	W =  90.000 deg,	P =   0.000 deg,	R =   90.000 deg
};
P[2097]{
   GP1:
	UF : 0, UT : 6,		CONFIG : 'N U T, 0, 0, 0',
	X =  98.445  mm,	Y =   -678.534  mm,	Z =   -242.195  mm,
	W =  90.000 deg,	P =   0.000 deg,	R =   90.000 deg
};
P[2098]{
   GP1:
	UF : 0, UT : 6,		CONFIG : 'N U T, 0, 0, 0',
	X =  104.284  mm,	Y =   -675.249  mm,	Z =   -241.987  mm,
	W =  90.000 deg,	P =   0.000 deg,	R =   90.000 deg
};
P[2099]{
   GP1:
	UF : 0, UT : 6,		CONFIG : 'N U T, 0, 0, 0',
	X =  105.353  mm,	Y =   -674.513  mm,	Z =   -242.274  mm,
	W =  90.000 deg,	P =   0.000 deg,	R =   90.000 deg
};
P[2100]{
   GP1:
	UF : 0, UT : 6,		CONFIG : 'N U T, 0, 0, 0',
	X =  107.366  mm,	Y =   -673.374  mm,	Z =   -242.215  mm,
	W =  90.000 deg,	P =   0.000 deg,	R =   90.000 deg
};
P[2101]{
   GP1:
	UF : 0, UT : 6,		CONFIG : 'N U T, 0, 0, 0',
	X =  110.303  mm,	Y =   -671.720  mm,	Z =   -242.116  mm,
	W =  90.000 deg,	P =   0.000 deg,	R =   90.000 deg
};
P[2102]{
   GP1:
	UF : 0, UT : 6,		CONFIG : 'N U T, 0, 0, 0',
	X =  111.391  mm,	Y =   -671.119  mm,	Z =   -242.049  mm,
	W =  90.000 deg,	P =   0.000 deg,	R =   90.000 deg
};
P[2103]{
   GP1:
	UF : 0, UT : 6,		CONFIG : 'N U T, 0, 0, 0',
	X =  113.149  mm,	Y =   -670.072  mm,	Z =   -242.125  mm,
	W =  90.000 deg,	P =   0.000 deg,	R =   90.000 deg
};
P[2104]{
   GP1:
	UF : 0, UT : 6,		CONFIG : 'N U T, 0, 0, 0',
	X =  114.405  mm,	Y =   -669.261  mm,	Z =   -242.337  mm,
	W =  90.000 deg,	P =   0.000 deg,	R =   90.000 deg
};
P[2105]{
   GP1:
	UF : 0, UT : 6,		CONFIG : 'N U T, 0, 0, 0',
	X =  118.642  mm,	Y =   -666.812  mm,	Z =   -242.340  mm,
	W =  90.000 deg,	P =   0.000 deg,	R =   90.000 deg
};
P[2106]{
   GP1:
	UF : 0, UT : 6,		CONFIG : 'N U T, 0, 0, 0',
	X =  119.817  mm,	Y =   -666.137  mm,	Z =   -242.334  mm,
	W =  90.000 deg,	P =   0.000 deg,	R =   90.000 deg
};
P[2107]{
   GP1:
	UF : 0, UT : 6,		CONFIG : 'N U T, 0, 0, 0',
	X =  120.600  mm,	Y =   -665.719  mm,	Z =   -242.251  mm,
	W =  90.000 deg,	P =   0.000 deg,	R =   90.000 deg
};
P[2108]{
   GP1:
	UF : 0, UT : 6,		CONFIG : 'N U T, 0, 0, 0',
	X =  123.719  mm,	Y =   -663.949  mm,	Z =   -242.176  mm,
	W =  90.000 deg,	P =   0.000 deg,	R =   90.000 deg
};
P[2109]{
   GP1:
	UF : 0, UT : 6,		CONFIG : 'N U T, 0, 0, 0',
	X =  125.494  mm,	Y =   -662.843  mm,	Z =   -242.374  mm,
	W =  90.000 deg,	P =   0.000 deg,	R =   90.000 deg
};
P[2110]{
   GP1:
	UF : 0, UT : 6,		CONFIG : 'N U T, 0, 0, 0',
	X =  129.879  mm,	Y =   -660.464  mm,	Z =   -242.003  mm,
	W =  90.000 deg,	P =   0.000 deg,	R =   90.000 deg
};
P[2111]{
   GP1:
	UF : 0, UT : 6,		CONFIG : 'N U T, 0, 0, 0',
	X =  132.744  mm,	Y =   -658.730  mm,	Z =   -242.195  mm,
	W =  90.000 deg,	P =   0.000 deg,	R =   90.000 deg
};
P[2112]{
   GP1:
	UF : 0, UT : 6,		CONFIG : 'N U T, 0, 0, 0',
	X =  134.698  mm,	Y =   -657.634  mm,	Z =   -242.116  mm,
	W =  90.000 deg,	P =   0.000 deg,	R =   90.000 deg
};
P[2113]{
   GP1:
	UF : 0, UT : 6,		CONFIG : 'N U T, 0, 0, 0',
	X =  135.518  mm,	Y =   -657.121  mm,	Z =   -242.214  mm,
	W =  90.000 deg,	P =   0.000 deg,	R =   90.000 deg
};
P[2114]{
   GP1:
	UF : 0, UT : 6,		CONFIG : 'N U T, 0, 0, 0',
	X =  143.347  mm,	Y =   -652.647  mm,	Z =   -242.099  mm,
	W =  90.000 deg,	P =   0.000 deg,	R =   90.000 deg
};
P[2115]{
   GP1:
	UF : 0, UT : 6,		CONFIG : 'N U T, 0, 0, 0',
	X =  144.078  mm,	Y =   -652.197  mm,	Z =   -242.167  mm,
	W =  90.000 deg,	P =   0.000 deg,	R =   90.000 deg
};
P[2116]{
   GP1:
	UF : 0, UT : 6,		CONFIG : 'N U T, 0, 0, 0',
	X =  145.223  mm,	Y =   -651.456  mm,	Z =   -242.362  mm,
	W =  90.000 deg,	P =   0.000 deg,	R =   90.000 deg
};
P[2117]{
   GP1:
	UF : 0, UT : 6,		CONFIG : 'N U T, 0, 0, 0',
	X =  149.521  mm,	Y =   -649.083  mm,	Z =   -242.100  mm,
	W =  90.000 deg,	P =   0.000 deg,	R =   90.000 deg
};
P[2118]{
   GP1:
	UF : 0, UT : 6,		CONFIG : 'N U T, 0, 0, 0',
	X =  150.339  mm,	Y =   -648.695  mm,	Z =   -241.893  mm,
	W =  90.000 deg,	P =   0.000 deg,	R =   90.000 deg
};
P[2119]{
   GP1:
	UF : 0, UT : 6,		CONFIG : 'N U T, 0, 0, 0',
	X =  151.021  mm,	Y =   -648.178  mm,	Z =   -242.192  mm,
	W =  90.000 deg,	P =   0.000 deg,	R =   90.000 deg
};
P[2120]{
   GP1:
	UF : 0, UT : 6,		CONFIG : 'N U T, 0, 0, 0',
	X =  152.713  mm,	Y =   -647.213  mm,	Z =   -242.164  mm,
	W =  90.000 deg,	P =   0.000 deg,	R =   90.000 deg
};
P[2121]{
   GP1:
	UF : 0, UT : 6,		CONFIG : 'N U T, 0, 0, 0',
	X =  153.696  mm,	Y =   -646.619  mm,	Z =   -242.228  mm,
	W =  90.000 deg,	P =   0.000 deg,	R =   90.000 deg
};
P[2122]{
   GP1:
	UF : 0, UT : 6,		CONFIG : 'N U T, 0, 0, 0',
	X =  154.593  mm,	Y =   -646.059  mm,	Z =   -242.330  mm,
	W =  90.000 deg,	P =   0.000 deg,	R =   90.000 deg
};
P[2123]{
   GP1:
	UF : 0, UT : 6,		CONFIG : 'N U T, 0, 0, 0',
	X =  158.846  mm,	Y =   -643.622  mm,	Z =   -242.287  mm,
	W =  90.000 deg,	P =   0.000 deg,	R =   90.000 deg
};
P[2124]{
   GP1:
	UF : 0, UT : 6,		CONFIG : 'N U T, 0, 0, 0',
	X =  161.233  mm,	Y =   -642.353  mm,	Z =   -242.021  mm,
	W =  90.000 deg,	P =   0.000 deg,	R =   90.000 deg
};
P[2125]{
   GP1:
	UF : 0, UT : 6,		CONFIG : 'N U T, 0, 0, 0',
	X =  164.420  mm,	Y =   -640.394  mm,	Z =   -242.307  mm,
	W =  90.000 deg,	P =   0.000 deg,	R =   90.000 deg
};
P[2126]{
   GP1:
	UF : 0, UT : 6,		CONFIG : 'N U T, 0, 0, 0',
	X =  166.261  mm,	Y =   -639.330  mm,	Z =   -242.311  mm,
	W =  90.000 deg,	P =   0.000 deg,	R =   90.000 deg
};
P[2127]{
   GP1:
	UF : 0, UT : 6,		CONFIG : 'N U T, 0, 0, 0',
	X =  166.963  mm,	Y =   -639.005  mm,	Z =   -242.115  mm,
	W =  90.000 deg,	P =   0.000 deg,	R =   90.000 deg
};
P[2128]{
   GP1:
	UF : 0, UT : 6,		CONFIG : 'N U T, 0, 0, 0',
	X =  169.189  mm,	Y =   -637.626  mm,	Z =   -242.343  mm,
	W =  90.000 deg,	P =   0.000 deg,	R =   90.000 deg
};
P[2129]{
   GP1:
	UF : 0, UT : 6,		CONFIG : 'N U T, 0, 0, 0',
	X =  170.609  mm,	Y =   -636.897  mm,	Z =   -242.124  mm,
	W =  90.000 deg,	P =   0.000 deg,	R =   90.000 deg
};
P[2130]{
   GP1:
	UF : 0, UT : 6,		CONFIG : 'N U T, 0, 0, 0',
	X =  173.140  mm,	Y =   -635.372  mm,	Z =   -242.276  mm,
	W =  90.000 deg,	P =   0.000 deg,	R =   90.000 deg
};
P[2131]{
   GP1:
	UF : 0, UT : 6,		CONFIG : 'N U T, 0, 0, 0',
	X =  176.589  mm,	Y =   -633.356  mm,	Z =   -242.335  mm,
	W =  90.000 deg,	P =   0.000 deg,	R =   90.000 deg
};
P[2132]{
   GP1:
	UF : 0, UT : 6,		CONFIG : 'N U T, 0, 0, 0',
	X =  179.057  mm,	Y =   -631.933  mm,	Z =   -242.332  mm,
	W =  90.000 deg,	P =   0.000 deg,	R =   90.000 deg
};
P[2133]{
   GP1:
	UF : 0, UT : 6,		CONFIG : 'N U T, 0, 0, 0',
	X =  181.582  mm,	Y =   -630.509  mm,	Z =   -242.251  mm,
	W =  90.000 deg,	P =   0.000 deg,	R =   90.000 deg
};
P[2134]{
   GP1:
	UF : 0, UT : 6,		CONFIG : 'N U T, 0, 0, 0',
	X =  183.130  mm,	Y =   -629.683  mm,	Z =   -242.086  mm,
	W =  90.000 deg,	P =   0.000 deg,	R =   90.000 deg
};
P[2135]{
   GP1:
	UF : 0, UT : 6,		CONFIG : 'N U T, 0, 0, 0',
	X =  184.824  mm,	Y =   -628.721  mm,	Z =   -242.048  mm,
	W =  90.000 deg,	P =   0.000 deg,	R =   90.000 deg
};
P[2136]{
   GP1:
	UF : 0, UT : 6,		CONFIG : 'N U T, 0, 0, 0',
	X =  186.772  mm,	Y =   -627.515  mm,	Z =   -242.244  mm,
	W =  90.000 deg,	P =   0.000 deg,	R =   90.000 deg
};
P[2137]{
   GP1:
	UF : 0, UT : 6,		CONFIG : 'N U T, 0, 0, 0',
	X =  188.247  mm,	Y =   -626.664  mm,	Z =   -242.241  mm,
	W =  90.000 deg,	P =   0.000 deg,	R =   90.000 deg
};
P[2138]{
   GP1:
	UF : 0, UT : 6,		CONFIG : 'N U T, 0, 0, 0',
	X =  192.750  mm,	Y =   -624.114  mm,	Z =   -242.121  mm,
	W =  90.000 deg,	P =   0.000 deg,	R =   90.000 deg
};
P[2139]{
   GP1:
	UF : 0, UT : 6,		CONFIG : 'N U T, 0, 0, 0',
	X =  193.446  mm,	Y =   -623.732  mm,	Z =   -242.070  mm,
	W =  90.000 deg,	P =   0.000 deg,	R =   90.000 deg
};
P[2140]{
   GP1:
	UF : 0, UT : 6,		CONFIG : 'N U T, 0, 0, 0',
	X =  195.025  mm,	Y =   -622.832  mm,	Z =   -242.044  mm,
	W =  90.000 deg,	P =   0.000 deg,	R =   90.000 deg
};
P[2141]{
   GP1:
	UF : 0, UT : 6,		CONFIG : 'N U T, 0, 0, 0',
	X =  197.669  mm,	Y =   -621.209  mm,	Z =   -242.278  mm,
	W =  90.000 deg,	P =   0.000 deg,	R =   90.000 deg
};
P[2142]{
   GP1:
	UF : 0, UT : 6,		CONFIG : 'N U T, 0, 0, 0',
	X =  199.485  mm,	Y =   -620.126  mm,	Z =   -242.361  mm,
	W =  90.000 deg,	P =   0.000 deg,	R =   90.000 deg
};
P[2143]{
   GP1:
	UF : 0, UT : 6,		CONFIG : 'N U T, 0, 0, 0',
	X =  200.341  mm,	Y =   -619.730  mm,	Z =   -242.123  mm,
	W =  90.000 deg,	P =   0.000 deg,	R =   90.000 deg
};
P[2144]{
   GP1:
	UF : 0, UT : 6,		CONFIG : 'N U T, 0, 0, 0',
	X =  203.567  mm,	Y =   -617.892  mm,	Z =   -242.063  mm,
	W =  90.000 deg,	P =   0.000 deg,	R =   90.000 deg
};
P[2145]{
   GP1:
	UF : 0, UT : 6,		CONFIG : 'N U T, 0, 0, 0',
	X =  208.016  mm,	Y =   -615.308  mm,	Z =   -242.100  mm,
	W =  90.000 deg,	P =   0.000 deg,	R =   90.000 deg
};
P[2146]{
   GP1:
	UF : 0, UT : 6,		CONFIG : 'N U T, 0, 0, 0',
	X =  208.666  mm,	Y =   -615.001  mm,	Z =   -241.933  mm,
	W =  90.000 deg,	P =   0.000 deg,	R =   90.000 deg
};
P[2147]{
   GP1:
	UF : 0, UT : 6,		CONFIG : 'N U T, 0, 0, 0',
	X =  211.605  mm,	Y =   -613.307  mm,	Z =   -241.925  mm,
	W =  90.000 deg,	P =   0.000 deg,	R =   90.000 deg
};
P[2148]{
   GP1:
	UF : 0, UT : 6,		CONFIG : 'N U T, 0, 0, 0',
	X =  213.043  mm,	Y =   -612.321  mm,	Z =   -242.304  mm,
	W =  90.000 deg,	P =   0.000 deg,	R =   90.000 deg
};
P[2149]{
   GP1:
	UF : 0, UT : 6,		CONFIG : 'N U T, 0, 0, 0',
	X =  213.786  mm,	Y =   -612.012  mm,	Z =   -242.013  mm,
	W =  90.000 deg,	P =   0.000 deg,	R =   90.000 deg
};
P[2150]{
   GP1:
	UF : 0, UT : 6,		CONFIG : 'N U T, 0, 0, 0',
	X =  217.019  mm,	Y =   -610.058  mm,	Z =   -242.225  mm,
	W =  90.000 deg,	P =   0.000 deg,	R =   90.000 deg
};
P[2151]{
   GP1:
	UF : 0, UT : 6,		CONFIG : 'N U T, 0, 0, 0',
	X =  217.928  mm,	Y =   -609.469  mm,	Z =   -242.381  mm,
	W =  90.000 deg,	P =   0.000 deg,	R =   90.000 deg
};
P[2152]{
   GP1:
	UF : 0, UT : 6,		CONFIG : 'N U T, 0, 0, 0',
	X =  220.660  mm,	Y =   -607.931  mm,	Z =   -242.286  mm,
	W =  90.000 deg,	P =   0.000 deg,	R =   90.000 deg
};
P[2153]{
   GP1:
	UF : 0, UT : 6,		CONFIG : 'N U T, 0, 0, 0',
	X =  222.324  mm,	Y =   -607.109  mm,	Z =   -241.947  mm,
	W =  90.000 deg,	P =   0.000 deg,	R =   90.000 deg
};
P[2154]{
   GP1:
	UF : 0, UT : 6,		CONFIG : 'N U T, 0, 0, 0',
	X =  223.722  mm,	Y =   -606.134  mm,	Z =   -242.357  mm,
	W =  90.000 deg,	P =   0.000 deg,	R =   90.000 deg
};
P[2155]{
   GP1:
	UF : 0, UT : 6,		CONFIG : 'N U T, 0, 0, 0',
	X =  227.232  mm,	Y =   -604.250  mm,	Z =   -242.009  mm,
	W =  90.000 deg,	P =   0.000 deg,	R =   90.000 deg
};
P[2156]{
   GP1:
	UF : 0, UT : 6,		CONFIG : 'N U T, 0, 0, 0',
	X =  229.183  mm,	Y =   -602.996  mm,	Z =   -242.322  mm,
	W =  90.000 deg,	P =   0.000 deg,	R =   90.000 deg
};
P[2157]{
   GP1:
	UF : 0, UT : 6,		CONFIG : 'N U T, 0, 0, 0',
	X =  230.455  mm,	Y =   -602.331  mm,	Z =   -242.152  mm,
	W =  90.000 deg,	P =   0.000 deg,	R =   90.000 deg
};
P[2158]{
   GP1:
	UF : 0, UT : 6,		CONFIG : 'N U T, 0, 0, 0',
	X =  231.314  mm,	Y =   -601.740  mm,	Z =   -242.380  mm,
	W =  90.000 deg,	P =   0.000 deg,	R =   90.000 deg
};
P[2159]{
   GP1:
	UF : 0, UT : 6,		CONFIG : 'N U T, 0, 0, 0',
	X =  232.191  mm,	Y =   -601.275  mm,	Z =   -242.279  mm,
	W =  90.000 deg,	P =   0.000 deg,	R =   90.000 deg
};
P[2160]{
   GP1:
	UF : 0, UT : 6,		CONFIG : 'N U T, 0, 0, 0',
	X =  233.158  mm,	Y =   -600.716  mm,	Z =   -242.281  mm,
	W =  90.000 deg,	P =   0.000 deg,	R =   90.000 deg
};
P[2161]{
   GP1:
	UF : 0, UT : 6,		CONFIG : 'N U T, 0, 0, 0',
	X =  235.314  mm,	Y =   -599.475  mm,	Z =   -242.271  mm,
	W =  90.000 deg,	P =   0.000 deg,	R =   90.000 deg
};
P[2162]{
   GP1:
	UF : 0, UT : 6,		CONFIG : 'N U T, 0, 0, 0',
	X =  236.403  mm,	Y =   -598.903  mm,	Z =   -242.135  mm,
	W =  90.000 deg,	P =   0.000 deg,	R =   90.000 deg
};
P[2163]{
   GP1:
	UF : 0, UT : 6,		CONFIG : 'N U T, 0, 0, 0',
	X =  238.414  mm,	Y =   -597.723  mm,	Z =   -242.183  mm,
	W =  90.000 deg,	P =   0.000 deg,	R =   90.000 deg
};
P[2164]{
   GP1:
	UF : 0, UT : 6,		CONFIG : 'N U T, 0, 0, 0',
	X =  244.113  mm,	Y =   -594.505  mm,	Z =   -242.004  mm,
	W =  90.000 deg,	P =   0.000 deg,	R =   90.000 deg
};
P[2165]{
   GP1:
	UF : 0, UT : 6,		CONFIG : 'N U T, 0, 0, 0',
	X =  246.683  mm,	Y =   -592.964  mm,	Z =   -242.143  mm,
	W =  90.000 deg,	P =   0.000 deg,	R =   90.000 deg
};
P[2166]{
   GP1:
	UF : 0, UT : 6,		CONFIG : 'N U T, 0, 0, 0',
	X =  247.661  mm,	Y =   -592.339  mm,	Z =   -242.291  mm,
	W =  90.000 deg,	P =   0.000 deg,	R =   90.000 deg
};
P[2167]{
   GP1:
	UF : 0, UT : 6,		CONFIG : 'N U T, 0, 0, 0',
	X =  248.771  mm,	Y =   -591.827  mm,	Z =   -241.978  mm,
	W =  90.000 deg,	P =   0.000 deg,	R =   90.000 deg
};
P[2168]{
   GP1:
	UF : 0, UT : 6,		CONFIG : 'N U T, 0, 0, 0',
	X =  251.090  mm,	Y =   -590.345  mm,	Z =   -242.325  mm,
	W =  90.000 deg,	P =   0.000 deg,	R =   90.000 deg
};
P[2169]{
   GP1:
	UF : 0, UT : 6,		CONFIG : 'N U T, 0, 0, 0',
	X =  251.938  mm,	Y =   -590.016  mm,	Z =   -241.934  mm,
	W =  90.000 deg,	P =   0.000 deg,	R =   90.000 deg
};
P[2170]{
   GP1:
	UF : 0, UT : 6,		CONFIG : 'N U T, 0, 0, 0',
	X =  255.560  mm,	Y =   -587.768  mm,	Z =   -242.316  mm,
	W =  90.000 deg,	P =   0.000 deg,	R =   90.000 deg
};
P[2171]{
   GP1:
	UF : 0, UT : 6,		CONFIG : 'N U T, 0, 0, 0',
	X =  257.010  mm,	Y =   -586.959  mm,	Z =   -242.248  mm,
	W =  90.000 deg,	P =   0.000 deg,	R =   90.000 deg
};
P[2172]{
   GP1:
	UF : 0, UT : 6,		CONFIG : 'N U T, 0, 0, 0',
	X =  258.469  mm,	Y =   -586.079  mm,	Z =   -242.337  mm,
	W =  90.000 deg,	P =   0.000 deg,	R =   90.000 deg
};
P[2173]{
   GP1:
	UF : 0, UT : 6,		CONFIG : 'N U T, 0, 0, 0',
	X =  262.285  mm,	Y =   -583.933  mm,	Z =   -242.198  mm,
	W =  90.000 deg,	P =   0.000 deg,	R =   90.000 deg
};
P[2174]{
   GP1:
	UF : 0, UT : 6,		CONFIG : 'N U T, 0, 0, 0',
	X =  265.570  mm,	Y =   -581.991  mm,	Z =   -242.309  mm,
	W =  90.000 deg,	P =   0.000 deg,	R =   90.000 deg
};
P[2175]{
   GP1:
	UF : 0, UT : 6,		CONFIG : 'N U T, 0, 0, 0',
	X =  267.214  mm,	Y =   -581.154  mm,	Z =   -242.036  mm,
	W =  90.000 deg,	P =   0.000 deg,	R =   90.000 deg
};
P[2176]{
   GP1:
	UF : 0, UT : 6,		CONFIG : 'N U T, 0, 0, 0',
	X =  269.085  mm,	Y =   -579.962  mm,	Z =   -242.306  mm,
	W =  90.000 deg,	P =   0.000 deg,	R =   90.000 deg
};
P[2177]{
   GP1:
	UF : 0, UT : 6,		CONFIG : 'N U T, 0, 0, 0',
	X =  271.474  mm,	Y =   -578.555  mm,	Z =   -242.373  mm,
	W =  90.000 deg,	P =   0.000 deg,	R =   90.000 deg
};
P[2178]{
   GP1:
	UF : 0, UT : 6,		CONFIG : 'N U T, 0, 0, 0',
	X =  273.966  mm,	Y =   -577.236  mm,	Z =   -242.081  mm,
	W =  90.000 deg,	P =   0.000 deg,	R =   90.000 deg
};
P[2179]{
   GP1:
	UF : 0, UT : 6,		CONFIG : 'N U T, 0, 0, 0',
	X =  277.153  mm,	Y =   -575.456  mm,	Z =   -241.936  mm,
	W =  90.000 deg,	P =   0.000 deg,	R =   90.000 deg
};
P[2180]{
   GP1:
	UF : 0, UT : 6,		CONFIG : 'N U T, 0, 0, 0',
	X =  284.062  mm,	Y =   -571.298  mm,	Z =   -242.346  mm,
	W =  90.000 deg,	P =   0.000 deg,	R =   90.000 deg
};
P[2181]{
   GP1:
	UF : 0, UT : 6,		CONFIG : 'N U T, 0, 0, 0',
	X =  284.968  mm,	Y =   -570.760  mm,	Z =   -242.381  mm,
	W =  90.000 deg,	P =   0.000 deg,	R =   90.000 deg
};
P[2182]{
   GP1:
	UF : 0, UT : 6,		CONFIG : 'N U T, 0, 0, 0',
	X =  285.824  mm,	Y =   -570.320  mm,	Z =   -242.251  mm,
	W =  90.000 deg,	P =   0.000 deg,	R =   90.000 deg
};
P[2183]{
   GP1:
	UF : 0, UT : 6,		CONFIG : 'N U T, 0, 0, 0',
	X =  286.911  mm,	Y =   -569.684  mm,	Z =   -242.272  mm,
	W =  90.000 deg,	P =   0.000 deg,	R =   90.000 deg
};
P[2184]{
   GP1:
	UF : 0, UT : 6,		CONFIG : 'N U T, 0, 0, 0',
	X =  290.019  mm,	Y =   -567.905  mm,	Z =   -242.233  mm,
	W =  90.000 deg,	P =   0.000 deg,	R =   90.000 deg
};
P[2185]{
   GP1:
	UF : 0, UT : 6,		CONFIG : 'N U T, 0, 0, 0',
	X =  292.325  mm,	Y =   -566.551  mm,	Z =   -242.287  mm,
	W =  90.000 deg,	P =   0.000 deg,	R =   90.000 deg
};
P[2186]{
   GP1:
	UF : 0, UT : 6,		CONFIG : 'N U T, 0, 0, 0',
	X =  294.546  mm,	Y =   -565.345  mm,	Z =   -242.103  mm,
	W =  90.000 deg,	P =   0.000 deg,	R =   90.000 deg
};
P[2187]{
   GP1:
	UF : 0, UT : 6,		CONFIG : 'N U T, 0, 0, 0',
	X =  296.447  mm,	Y =   -564.152  mm,	Z =   -242.334  mm,
	W =  90.000 deg,	P =   0.000 deg,	R =   90.000 deg
};
P[2188]{
   GP1:
	UF : 0, UT : 6,		CONFIG : 'N U T, 0, 0, 0',
	X =  299.729  mm,	Y =   -562.268  mm,	Z =   -242.306  mm,
	W =  90.000 deg,	P =   0.000 deg,	R =   90.000 deg
};
P[2189]{
   GP1:
	UF : 0, UT : 6,		CONFIG : 'N U T, 0, 0, 0',
	X =  301.875  mm,	Y =   -561.069  mm,	Z =   -242.211  mm,
	W =  90.000 deg,	P =   0.000 deg,	R =   90.000 deg
};
P[2190]{
   GP1:
	UF : 0, UT : 6,		CONFIG : 'N U T, 0, 0, 0',
	X =  303.015  mm,	Y =   -560.355  mm,	Z =   -242.345  mm,
	W =  90.000 deg,	P =   0.000 deg,	R =   90.000 deg
};
P[2191]{
   GP1:
	UF : 0, UT : 6,		CONFIG : 'N U T, 0, 0, 0',
	X =  303.649  mm,	Y =   -560.057  mm,	Z =   -242.180  mm,
	W =  90.000 deg,	P =   0.000 deg,	R =   90.000 deg
};
P[2192]{
   GP1:
	UF : 0, UT : 6,		CONFIG : 'N U T, 0, 0, 0',
	X =  307.343  mm,	Y =   -557.958  mm,	Z =   -242.099  mm,
	W =  90.000 deg,	P =   0.000 deg,	R =   90.000 deg
};
P[2193]{
   GP1:
	UF : 0, UT : 6,		CONFIG : 'N U T, 0, 0, 0',
	X =  307.941  mm,	Y =   -557.528  mm,	Z =   -242.305  mm,
	W =  90.000 deg,	P =   0.000 deg,	R =   90.000 deg
};
P[2194]{
   GP1:
	UF : 0, UT : 6,		CONFIG : 'N U T, 0, 0, 0',
	X =  309.717  mm,	Y =   -556.576  mm,	Z =   -242.127  mm,
	W =  90.000 deg,	P =   0.000 deg,	R =   90.000 deg
};
P[2195]{
   GP1:
	UF : 0, UT : 6,		CONFIG : 'N U T, 0, 0, 0',
	X =  312.318  mm,	Y =   -555.012  mm,	Z =   -242.277  mm,
	W =  90.000 deg,	P =   0.000 deg,	R =   90.000 deg
};
P[2196]{
   GP1:
	UF : 0, UT : 6,		CONFIG : 'N U T, 0, 0, 0',
	X =  314.668  mm,	Y =   -553.723  mm,	Z =   -242.112  mm,
	W =  90.000 deg,	P =   0.000 deg,	R =   90.000 deg
};
P[2197]{
   GP1:
	UF : 0, UT : 6,		CONFIG : 'N U T, 0, 0, 0',
	X =  316.747  mm,	Y =   -552.451  mm,	Z =   -242.286  mm,
	W =  90.000 deg,	P =   0.000 deg,	R =   90.000 deg
};
P[2198]{
   GP1:
	UF : 0, UT : 6,		CONFIG : 'N U T, 0, 0, 0',
	X =  320.566  mm,	Y =   -550.313  mm,	Z =   -242.124  mm,
	W =  90.000 deg,	P =   0.000 deg,	R =   90.000 deg
};
P[2199]{
   GP1:
	UF : 0, UT : 6,		CONFIG : 'N U T, 0, 0, 0',
	X =  322.324  mm,	Y =   -549.263  mm,	Z =   -242.209  mm,
	W =  90.000 deg,	P =   0.000 deg,	R =   90.000 deg
};
P[2200]{
   GP1:
	UF : 0, UT : 6,		CONFIG : 'N U T, 0, 0, 0',
	X =  323.434  mm,	Y =   -548.597  mm,	Z =   -242.269  mm,
	W =  90.000 deg,	P =   0.000 deg,	R =   90.000 deg
};
P[2201]{
   GP1:
	UF : 0, UT : 6,		CONFIG : 'N U T, 0, 0, 0',
	X =  325.084  mm,	Y =   -547.599  mm,	Z =   -242.377  mm,
	W =  90.000 deg,	P =   0.000 deg,	R =   90.000 deg
};
P[2202]{
   GP1:
	UF : 0, UT : 6,		CONFIG : 'N U T, 0, 0, 0',
	X =  327.231  mm,	Y =   -546.494  mm,	Z =   -242.053  mm,
	W =  90.000 deg,	P =   0.000 deg,	R =   90.000 deg
};
P[2203]{
   GP1:
	UF : 0, UT : 6,		CONFIG : 'N U T, 0, 0, 0',
	X =  329.018  mm,	Y =   -545.380  mm,	Z =   -242.251  mm,
	W =  90.000 deg,	P =   0.000 deg,	R =   90.000 deg
};
P[2204]{
   GP1:
	UF : 0, UT : 6,		CONFIG : 'N U T, 0, 0, 0',
	X =  331.852  mm,	Y =   -543.709  mm,	Z =   -242.335  mm,
	W =  90.000 deg,	P =   0.000 deg,	R =   90.000 deg
};
P[2205]{
   GP1:
	UF : 0, UT : 6,		CONFIG : 'N U T, 0, 0, 0',
	X =  333.451  mm,	Y =   -542.914  mm,	Z =   -242.024  mm,
	W =  90.000 deg,	P =   0.000 deg,	R =   90.000 deg
};
P[2206]{
   GP1:
	UF : 0, UT : 6,		CONFIG : 'N U T, 0, 0, 0',
	X =  339.237  mm,	Y =   -539.581  mm,	Z =   -242.005  mm,
	W =  90.000 deg,	P =   0.000 deg,	R =   90.000 deg
};
P[2207]{
   GP1:
	UF : 0, UT : 6,		CONFIG : 'N U T, 0, 0, 0',
	X =  341.023  mm,	Y =   -538.535  mm,	Z =   -242.042  mm,
	W =  90.000 deg,	P =   0.000 deg,	R =   90.000 deg
};
P[2208]{
   GP1:
	UF : 0, UT : 6,		CONFIG : 'N U T, 0, 0, 0',
	X =  342.474  mm,	Y =   -537.737  mm,	Z =   -241.944  mm,
	W =  90.000 deg,	P =   0.000 deg,	R =   90.000 deg
};
P[2209]{
   GP1:
	UF : 0, UT : 6,		CONFIG : 'N U T, 0, 0, 0',
	X =  343.347  mm,	Y =   -537.088  mm,	Z =   -242.296  mm,
	W =  90.000 deg,	P =   0.000 deg,	R =   90.000 deg
};
P[2210]{
   GP1:
	UF : 0, UT : 6,		CONFIG : 'N U T, 0, 0, 0',
	X =  346.299  mm,	Y =   -535.366  mm,	Z =   -242.340  mm,
	W =  90.000 deg,	P =   0.000 deg,	R =   90.000 deg
};
P[2211]{
   GP1:
	UF : 0, UT : 6,		CONFIG : 'N U T, 0, 0, 0',
	X =  350.272  mm,	Y =   -533.145  mm,	Z =   -242.163  mm,
	W =  90.000 deg,	P =   0.000 deg,	R =   90.000 deg
};
P[2212]{
   GP1:
	UF : 0, UT : 6,		CONFIG : 'N U T, 0, 0, 0',
	X =  352.462  mm,	Y =   -531.906  mm,	Z =   -242.102  mm,
	W =  90.000 deg,	P =   0.000 deg,	R =   90.000 deg
};
P[2213]{
   GP1:
	UF : 0, UT : 6,		CONFIG : 'N U T, 0, 0, 0',
	X =  354.304  mm,	Y =   -530.901  mm,	Z =   -241.958  mm,
	W =  90.000 deg,	P =   0.000 deg,	R =   90.000 deg
};
P[2214]{
   GP1:
	UF : 0, UT : 6,		CONFIG : 'N U T, 0, 0, 0',
	X =  357.314  mm,	Y =   -529.181  mm,	Z =   -241.916  mm,
	W =  90.000 deg,	P =   0.000 deg,	R =   90.000 deg
};
P[2215]{
   GP1:
	UF : 0, UT : 6,		CONFIG : 'N U T, 0, 0, 0',
	X =  359.415  mm,	Y =   -527.809  mm,	Z =   -242.300  mm,
	W =  90.000 deg,	P =   0.000 deg,	R =   90.000 deg
};
P[2216]{
   GP1:
	UF : 0, UT : 6,		CONFIG : 'N U T, 0, 0, 0',
	X =  361.903  mm,	Y =   -526.366  mm,	Z =   -242.314  mm,
	W =  90.000 deg,	P =   0.000 deg,	R =   90.000 deg
};
P[2217]{
   GP1:
	UF : 0, UT : 6,		CONFIG : 'N U T, 0, 0, 0',
	X =  363.917  mm,	Y =   -525.208  mm,	Z =   -242.302  mm,
	W =  90.000 deg,	P =   0.000 deg,	R =   90.000 deg
};
P[2218]{
   GP1:
	UF : 0, UT : 6,		CONFIG : 'N U T, 0, 0, 0',
	X =  367.035  mm,	Y =   -523.470  mm,	Z =   -242.155  mm,
	W =  90.000 deg,	P =   0.000 deg,	R =   90.000 deg
};
P[2219]{
   GP1:
	UF : 0, UT : 6,		CONFIG : 'N U T, 0, 0, 0',
	X =  370.243  mm,	Y =   -521.688  mm,	Z =   -241.981  mm,
	W =  90.000 deg,	P =   0.000 deg,	R =   90.000 deg
};
P[2220]{
   GP1:
	UF : 0, UT : 6,		CONFIG : 'N U T, 0, 0, 0',
	X =  372.116  mm,	Y =   -520.459  mm,	Z =   -242.340  mm,
	W =  90.000 deg,	P =   0.000 deg,	R =   90.000 deg
};
P[2221]{
   GP1:
	UF : 0, UT : 6,		CONFIG : 'N U T, 0, 0, 0',
	X =  374.384  mm,	Y =   -519.194  mm,	Z =   -242.233  mm,
	W =  90.000 deg,	P =   0.000 deg,	R =   90.000 deg
};
P[2222]{
   GP1:
	UF : 0, UT : 6,		CONFIG : 'N U T, 0, 0, 0',
	X =  377.428  mm,	Y =   -517.573  mm,	Z =   -241.902  mm,
	W =  90.000 deg,	P =   0.000 deg,	R =   90.000 deg
};
P[2223]{
   GP1:
	UF : 0, UT : 6,		CONFIG : 'N U T, 0, 0, 0',
	X =  379.034  mm,	Y =   -516.475  mm,	Z =   -242.315  mm,
	W =  90.000 deg,	P =   0.000 deg,	R =   90.000 deg
};
P[2224]{
   GP1:
	UF : 0, UT : 6,		CONFIG : 'N U T, 0, 0, 0',
	X =  383.186  mm,	Y =   -514.056  mm,	Z =   -242.368  mm,
	W =  90.000 deg,	P =   0.000 deg,	R =   90.000 deg
};
P[2225]{
   GP1:
	UF : 0, UT : 6,		CONFIG : 'N U T, 0, 0, 0',
	X =  384.076  mm,	Y =   -513.680  mm,	Z =   -242.032  mm,
	W =  90.000 deg,	P =   0.000 deg,	R =   90.000 deg
};
P[2226]{
   GP1:
	UF : 0, UT : 6,		CONFIG : 'N U T, 0, 0, 0',
	X =  388.801  mm,	Y =   -510.854  mm,	Z =   -242.268  mm,
	W =  90.000 deg,	P =   0.000 deg,	R =   90.000 deg
};
P[2227]{
   GP1:
	UF : 0, UT : 6,		CONFIG : 'N U T, 0, 0, 0',
	X =  389.435  mm,	Y =   -510.476  mm,	Z =   -242.300  mm,
	W =  90.000 deg,	P =   0.000 deg,	R =   90.000 deg
};
P[2228]{
   GP1:
	UF : 0, UT : 6,		CONFIG : 'N U T, 0, 0, 0',
	X =  390.253  mm,	Y =   -510.133  mm,	Z =   -241.986  mm,
	W =  90.000 deg,	P =   0.000 deg,	R =   90.000 deg
};
P[2229]{
   GP1:
	UF : 0, UT : 6,		CONFIG : 'N U T, 0, 0, 0',
	X =  392.120  mm,	Y =   -509.036  mm,	Z =   -242.034  mm,
	W =  90.000 deg,	P =   0.000 deg,	R =   90.000 deg
};
P[2230]{
   GP1:
	UF : 0, UT : 6,		CONFIG : 'N U T, 0, 0, 0',
	X =  393.408  mm,	Y =   -508.148  mm,	Z =   -242.382  mm,
	W =  90.000 deg,	P =   0.000 deg,	R =   90.000 deg
};
P[2231]{
   GP1:
	UF : 0, UT : 6,		CONFIG : 'N U T, 0, 0, 0',
	X =  396.863  mm,	Y =   -506.269  mm,	Z =   -242.101  mm,
	W =  90.000 deg,	P =   0.000 deg,	R =   90.000 deg
};
P[2232]{
   GP1:
	UF : 0, UT : 6,		CONFIG : 'N U T, 0, 0, 0',
	X =  399.660  mm,	Y =   -504.730  mm,	Z =   -241.918  mm,
	W =  90.000 deg,	P =   0.000 deg,	R =   90.000 deg
};
P[2233]{
   GP1:
	UF : 0, UT : 6,		CONFIG : 'N U T, 0, 0, 0',
	X =  400.293  mm,	Y =   -504.272  mm,	Z =   -242.139  mm,
	W =  90.000 deg,	P =   0.000 deg,	R =   90.000 deg
};
P[2234]{
   GP1:
	UF : 0, UT : 6,		CONFIG : 'N U T, 0, 0, 0',
	X =  401.370  mm,	Y =   -503.613  mm,	Z =   -242.231  mm,
	W =  90.000 deg,	P =   0.000 deg,	R =   90.000 deg
};
P[2235]{
   GP1:
	UF : 0, UT : 6,		CONFIG : 'N U T, 0, 0, 0',
	X =  407.087  mm,	Y =   -500.404  mm,	Z =   -242.007  mm,
	W =  90.000 deg,	P =   0.000 deg,	R =   90.000 deg
};
P[2236]{
   GP1:
	UF : 0, UT : 6,		CONFIG : 'N U T, 0, 0, 0',
	X =  408.943  mm,	Y =   -499.184  mm,	Z =   -242.367  mm,
	W =  90.000 deg,	P =   0.000 deg,	R =   90.000 deg
};
P[2237]{
   GP1:
	UF : 0, UT : 6,		CONFIG : 'N U T, 0, 0, 0',
	X =  409.656  mm,	Y =   -498.783  mm,	Z =   -242.344  mm,
	W =  90.000 deg,	P =   0.000 deg,	R =   90.000 deg
};
P[2238]{
   GP1:
	UF : 0, UT : 6,		CONFIG : 'N U T, 0, 0, 0',
	X =  411.200  mm,	Y =   -497.965  mm,	Z =   -242.164  mm,
	W =  90.000 deg,	P =   0.000 deg,	R =   90.000 deg
};
P[2239]{
   GP1:
	UF : 0, UT : 6,		CONFIG : 'N U T, 0, 0, 0',
	X =  414.821  mm,	Y =   -495.976  mm,	Z =   -241.919  mm,
	W =  90.000 deg,	P =   0.000 deg,	R =   90.000 deg
};
P[2240]{
   GP1:
	UF : 0, UT : 6,		CONFIG : 'N U T, 0, 0, 0',
	X =  415.662  mm,	Y =   -495.337  mm,	Z =   -242.288  mm,
	W =  90.000 deg,	P =   0.000 deg,	R =   90.000 deg
};
P[2241]{
   GP1:
	UF : 0, UT : 6,		CONFIG : 'N U T, 0, 0, 0',
	X =  416.850  mm,	Y =   -494.710  mm,	Z =   -242.147  mm,
	W =  90.000 deg,	P =   0.000 deg,	R =   90.000 deg
};
P[2242]{
   GP1:
	UF : 0, UT : 6,		CONFIG : 'N U T, 0, 0, 0',
	X =  420.083  mm,	Y =   -492.856  mm,	Z =   -242.115  mm,
	W =  90.000 deg,	P =   0.000 deg,	R =   90.000 deg
};
P[2243]{
   GP1:
	UF : 0, UT : 6,		CONFIG : 'N U T, 0, 0, 0',
	X =  420.759  mm,	Y =   -492.389  mm,	Z =   -242.302  mm,
	W =  90.000 deg,	P =   0.000 deg,	R =   90.000 deg
};
P[2244]{
   GP1:
	UF : 0, UT : 6,		CONFIG : 'N U T, 0, 0, 0',
	X =  422.736  mm,	Y =   -491.303  mm,	Z =   -242.166  mm,
	W =  90.000 deg,	P =   0.000 deg,	R =   90.000 deg
};
P[2245]{
   GP1:
	UF : 0, UT : 6,		CONFIG : 'N U T, 0, 0, 0',
	X =  423.883  mm,	Y =   -490.551  mm,	Z =   -242.385  mm,
	W =  90.000 deg,	P =   0.000 deg,	R =   90.000 deg
};
P[2246]{
   GP1:
	UF : 0, UT : 6,		CONFIG : 'N U T, 0, 0, 0',
	X =  425.632  mm,	Y =   -489.645  mm,	Z =   -242.131  mm,
	W =  90.000 deg,	P =   0.000 deg,	R =   90.000 deg
};
P[2247]{
   GP1:
	UF : 0, UT : 6,		CONFIG : 'N U T, 0, 0, 0',
	X =  430.039  mm,	Y =   -487.131  mm,	Z =   -242.059  mm,
	W =  90.000 deg,	P =   0.000 deg,	R =   90.000 deg
};
P[2248]{
   GP1:
	UF : 0, UT : 6,		CONFIG : 'N U T, 0, 0, 0',
	X =  430.777  mm,	Y =   -486.600  mm,	Z =   -242.313  mm,
	W =  90.000 deg,	P =   0.000 deg,	R =   90.000 deg
};
P[2249]{
   GP1:
	UF : 0, UT : 6,		CONFIG : 'N U T, 0, 0, 0',
	X =  434.490  mm,	Y =   -484.518  mm,	Z =   -242.161  mm,
	W =  90.000 deg,	P =   0.000 deg,	R =   90.000 deg
};
P[2250]{
   GP1:
	UF : 0, UT : 6,		CONFIG : 'N U T, 0, 0, 0',
	X =  435.101  mm,	Y =   -484.138  mm,	Z =   -242.227  mm,
	W =  90.000 deg,	P =   0.000 deg,	R =   90.000 deg
};
P[2251]{
   GP1:
	UF : 0, UT : 6,		CONFIG : 'N U T, 0, 0, 0',
	X =  439.075  mm,	Y =   -481.925  mm,	Z =   -242.029  mm,
	W =  90.000 deg,	P =   0.000 deg,	R =   90.000 deg
};
P[2252]{
   GP1:
	UF : 0, UT : 6,		CONFIG : 'N U T, 0, 0, 0',
	X =  440.112  mm,	Y =   -481.282  mm,	Z =   -242.137  mm,
	W =  90.000 deg,	P =   0.000 deg,	R =   90.000 deg
};
P[2253]{
   GP1:
	UF : 0, UT : 6,		CONFIG : 'N U T, 0, 0, 0',
	X =  444.811  mm,	Y =   -478.526  mm,	Z =   -242.243  mm,
	W =  90.000 deg,	P =   0.000 deg,	R =   90.000 deg
};
P[2254]{
   GP1:
	UF : 0, UT : 6,		CONFIG : 'N U T, 0, 0, 0',
	X =  445.758  mm,	Y =   -478.019  mm,	Z =   -242.146  mm,
	W =  90.000 deg,	P =   0.000 deg,	R =   90.000 deg
};
P[2255]{
   GP1:
	UF : 0, UT : 6,		CONFIG : 'N U T, 0, 0, 0',
	X =  447.036  mm,	Y =   -477.186  mm,	Z =   -242.377  mm,
	W =  90.000 deg,	P =   0.000 deg,	R =   90.000 deg
};
P[2256]{
   GP1:
	UF : 0, UT : 6,		CONFIG : 'N U T, 0, 0, 0',
	X =  450.885  mm,	Y =   -474.972  mm,	Z =   -242.357  mm,
	W =  90.000 deg,	P =   0.000 deg,	R =   90.000 deg
};
P[2257]{
   GP1:
	UF : 0, UT : 6,		CONFIG : 'N U T, 0, 0, 0',
	X =  453.570  mm,	Y =   -473.410  mm,	Z =   -242.385  mm,
	W =  90.000 deg,	P =   0.000 deg,	R =   90.000 deg
};
P[2258]{
   GP1:
	UF : 0, UT : 6,		CONFIG : 'N U T, 0, 0, 0',
	X =  454.575  mm,	Y =   -472.990  mm,	Z =   -241.995  mm,
	W =  90.000 deg,	P =   0.000 deg,	R =   90.000 deg
};
P[2259]{
   GP1:
	UF : 0, UT : 6,		CONFIG : 'N U T, 0, 0, 0',
	X =  455.439  mm,	Y =   -472.428  mm,	Z =   -242.148  mm,
	W =  90.000 deg,	P =   0.000 deg,	R =   90.000 deg
};
P[2260]{
   GP1:
	UF : 0, UT : 6,		CONFIG : 'N U T, 0, 0, 0',
	X =  460.724  mm,	Y =   -469.380  mm,	Z =   -242.141  mm,
	W =  90.000 deg,	P =   0.000 deg,	R =   90.000 deg
};
P[2261]{
   GP1:
	UF : 0, UT : 6,		CONFIG : 'N U T, 0, 0, 0',
	X =  461.291  mm,	Y =   -468.962  mm,	Z =   -242.360  mm,
	W =  90.000 deg,	P =   0.000 deg,	R =   90.000 deg
};
P[2262]{
   GP1:
	UF : 0, UT : 6,		CONFIG : 'N U T, 0, 0, 0',
	X =  463.577  mm,	Y =   -467.802  mm,	Z =   -241.973  mm,
	W =  90.000 deg,	P =   0.000 deg,	R =   90.000 deg
};
P[2263]{
   GP1:
	UF : 0, UT : 6,		CONFIG : 'N U T, 0, 0, 0',
	X =  464.292  mm,	Y =   -467.293  mm,	Z =   -242.206  mm,
	W =  90.000 deg,	P =   0.000 deg,	R =   90.000 deg
};
P[2264]{
   GP1:
	UF : 0, UT : 6,		CONFIG : 'N U T, 0, 0, 0',
	X =  468.302  mm,	Y =   -464.916  mm,	Z =   -242.353  mm,
	W =  90.000 deg,	P =   0.000 deg,	R =   90.000 deg
};
P[2265]{
   GP1:
	UF : 0, UT : 6,		CONFIG : 'N U T, 0, 0, 0',
	X =  469.058  mm,	Y =   -464.649  mm,	Z =   -241.943  mm,
	W =  90.000 deg,	P =   0.000 deg,	R =   90.000 deg
};
P[2266]{
   GP1:
	UF : 0, UT : 6,		CONFIG : 'N U T, 0, 0, 0',
	X =  472.753  mm,	Y =   -462.407  mm,	Z =   -242.205  mm,
	W =  90.000 deg,	P =   0.000 deg,	R =   90.000 deg
};
P[2267]{
   GP1:
	UF : 0, UT : 6,		CONFIG : 'N U T, 0, 0, 0',
	X =  473.970  mm,	Y =   -461.742  mm,	Z =   -242.115  mm,
	W =  90.000 deg,	P =   0.000 deg,	R =   90.000 deg
};
P[2268]{
   GP1:
	UF : 0, UT : 6,		CONFIG : 'N U T, 0, 0, 0',
	X =  476.365  mm,	Y =   -460.353  mm,	Z =   -242.129  mm,
	W =  90.000 deg,	P =   0.000 deg,	R =   90.000 deg
};
P[2269]{
   GP1:
	UF : 0, UT : 6,		CONFIG : 'N U T, 0, 0, 0',
	X =  478.299  mm,	Y =   -459.291  mm,	Z =   -242.000  mm,
	W =  90.000 deg,	P =   0.000 deg,	R =   90.000 deg
};
P[2270]{
   GP1:
	UF : 0, UT : 6,		CONFIG : 'N U T, 0, 0, 0',
	X =  479.109  mm,	Y =   -458.674  mm,	Z =   -242.361  mm,
	W =  90.000 deg,	P =   0.000 deg,	R =   90.000 deg
};
P[2271]{
   GP1:
	UF : 0, UT : 6,		CONFIG : 'N U T, 0, 0, 0',
	X =  484.841  mm,	Y =   -455.463  mm,	Z =   -242.121  mm,
	W =  90.000 deg,	P =   0.000 deg,	R =   90.000 deg
};
P[2272]{
   GP1:
	UF : 0, UT : 6,		CONFIG : 'N U T, 0, 0, 0',
	X =  486.890  mm,	Y =   -454.186  mm,	Z =   -242.349  mm,
	W =  90.000 deg,	P =   0.000 deg,	R =   90.000 deg
};
P[2273]{
   GP1:
	UF : 0, UT : 6,		CONFIG : 'N U T, 0, 0, 0',
	X =  492.068  mm,	Y =   -451.277  mm,	Z =   -242.153  mm,
	W =  90.000 deg,	P =   0.000 deg,	R =   90.000 deg
};
P[2274]{
   GP1:
	UF : 0, UT : 6,		CONFIG : 'N U T, 0, 0, 0',
	X =  492.694  mm,	Y =   -450.876  mm,	Z =   -242.250  mm,
	W =  90.000 deg,	P =   0.000 deg,	R =   90.000 deg
};
P[2275]{
   GP1:
	UF : 0, UT : 6,		CONFIG : 'N U T, 0, 0, 0',
	X =  495.587  mm,	Y =   -449.332  mm,	Z =   -241.942  mm,
	W =  90.000 deg,	P =   0.000 deg,	R =   90.000 deg
};
P[2276]{
   GP1:
	UF : 0, UT : 6,		CONFIG : 'N U T, 0, 0, 0',
	X =  496.136  mm,	Y =   -448.834  mm,	Z =   -242.381  mm,
	W =  90.000 deg,	P =   0.000 deg,	R =   90.000 deg
};
P[2277]{
   GP1:
	UF : 0, UT : 6,		CONFIG : 'N U T, 0, 0, 0',
	X =  497.108  mm,	Y =   -448.415  mm,	Z =   -242.034  mm,
	W =  90.000 deg,	P =   0.000 deg,	R =   90.000 deg
};
P[2278]{
   GP1:
	UF : 0, UT : 6,		CONFIG : 'N U T, 0, 0, 0',
	X =  498.207  mm,	Y =   -447.674  mm,	Z =   -242.294  mm,
	W =  90.000 deg,	P =   0.000 deg,	R =   90.000 deg
};
P[2279]{
   GP1:
	UF : 0, UT : 6,		CONFIG : 'N U T, 0, 0, 0',
	X =  500.155  mm,	Y =   -446.642  mm,	Z =   -242.070  mm,
	W =  90.000 deg,	P =   0.000 deg,	R =   90.000 deg
};
P[2280]{
   GP1:
	UF : 0, UT : 6,		CONFIG : 'N U T, 0, 0, 0',
	X =  501.066  mm,	Y =   -446.050  mm,	Z =   -242.229  mm,
	W =  90.000 deg,	P =   0.000 deg,	R =   90.000 deg
};
P[2281]{
   GP1:
	UF : 0, UT : 6,		CONFIG : 'N U T, 0, 0, 0',
	X =  502.720  mm,	Y =   -445.073  mm,	Z =   -242.283  mm,
	W =  90.000 deg,	P =   0.000 deg,	R =   90.000 deg
};
P[2282]{
   GP1:
	UF : 0, UT : 6,		CONFIG : 'N U T, 0, 0, 0',
	X =  506.089  mm,	Y =   -443.242  mm,	Z =   -242.005  mm,
	W =  90.000 deg,	P =   0.000 deg,	R =   90.000 deg
};
P[2283]{
   GP1:
	UF : 0, UT : 6,		CONFIG : 'N U T, 0, 0, 0',
	X =  506.760  mm,	Y =   -442.711  mm,	Z =   -242.354  mm,
	W =  90.000 deg,	P =   0.000 deg,	R =   90.000 deg
};
P[2284]{
   GP1:
	UF : 0, UT : 6,		CONFIG : 'N U T, 0, 0, 0',
	X =  508.006  mm,	Y =   -442.132  mm,	Z =   -242.015  mm,
	W =  90.000 deg,	P =   0.000 deg,	R =   90.000 deg
};
P[2285]{
   GP1:
	UF : 0, UT : 6,		CONFIG : 'N U T, 0, 0, 0',
	X =  508.908  mm,	Y =   -441.503  mm,	Z =   -242.277  mm,
	W =  90.000 deg,	P =   0.000 deg,	R =   90.000 deg
};
P[2286]{
   GP1:
	UF : 0, UT : 6,		CONFIG : 'N U T, 0, 0, 0',
	X =  511.832  mm,	Y =   -439.832  mm,	Z =   -242.234  mm,
	W =  90.000 deg,	P =   0.000 deg,	R =   90.000 deg
};
P[2287]{
   GP1:
	UF : 0, UT : 6,		CONFIG : 'N U T, 0, 0, 0',
	X =  512.918  mm,	Y =   -439.221  mm,	Z =   -242.194  mm,
	W =  90.000 deg,	P =   0.000 deg,	R =   90.000 deg
};
P[2288]{
   GP1:
	UF : 0, UT : 6,		CONFIG : 'N U T, 0, 0, 0',
	X =  514.896  mm,	Y =   -438.102  mm,	Z =   -242.140  mm,
	W =  90.000 deg,	P =   0.000 deg,	R =   90.000 deg
};
P[2289]{
   GP1:
	UF : 0, UT : 6,		CONFIG : 'N U T, 0, 0, 0',
	X =  517.100  mm,	Y =   -436.755  mm,	Z =   -242.319  mm,
	W =  90.000 deg,	P =   0.000 deg,	R =   90.000 deg
};
P[2290]{
   GP1:
	UF : 0, UT : 6,		CONFIG : 'N U T, 0, 0, 0',
	X =  518.516  mm,	Y =   -436.076  mm,	Z =   -241.983  mm,
	W =  90.000 deg,	P =   0.000 deg,	R =   90.000 deg
};
P[2291]{
   GP1:
	UF : 0, UT : 6,		CONFIG : 'N U T, 0, 0, 0',
	X =  523.189  mm,	Y =   -432.336  mm,	Z =   -242.185  mm,
	W =  90.000 deg,	P =   0.000 deg,	R =   90.000 deg
};
P[2292]{
   GP1:
	UF : 0, UT : 6,		CONFIG : 'N U T, 0, 0, 0',
	X =  525.786  mm,	Y =   -427.834  mm,	Z =   -242.200  mm,
	W =  90.000 deg,	P =   0.000 deg,	R =   90.000 deg
};
P[2293]{
   GP1:
	UF : 0, UT : 6,		CONFIG : 'N U T, 0, 0, 0',
	X =  525.657  mm,	Y =   -418.787  mm,	Z =   -242.012  mm,
	W =  90.000 deg,	P =   0.000 deg,	R =   90.000 deg
};
P[2294]{
   GP1:
	UF : 0, UT : 6,		CONFIG : 'N U T, 0, 0, 0',
	X =  525.109  mm,	Y =   -417.659  mm,	Z =   -242.107  mm,
	W =  90.000 deg,	P =   0.000 deg,	R =   90.000 deg
};
P[2295]{
   GP1:
	UF : 0, UT : 6,		CONFIG : 'N U T, 0, 0, 0',
	X =  524.700  mm,	Y =   -416.910  mm,	Z =   -242.252  mm,
	W =  90.000 deg,	P =   0.000 deg,	R =   90.000 deg
};
P[2296]{
   GP1:
	UF : 0, UT : 6,		CONFIG : 'N U T, 0, 0, 0',
	X =  523.461  mm,	Y =   -414.433  mm,	Z =   -241.907  mm,
	W =  90.000 deg,	P =   0.000 deg,	R =   90.000 deg
};
P[2297]{
   GP1:
	UF : 0, UT : 6,		CONFIG : 'N U T, 0, 0, 0',
	X =  522.163  mm,	Y =   -412.520  mm,	Z =   -242.375  mm,
	W =  90.000 deg,	P =   0.000 deg,	R =   90.000 deg
};
P[2298]{
   GP1:
	UF : 0, UT : 6,		CONFIG : 'N U T, 0, 0, 0',
	X =  521.014  mm,	Y =   -410.195  mm,	Z =   -241.907  mm,
	W =  90.000 deg,	P =   0.000 deg,	R =   90.000 deg
};
P[2299]{
   GP1:
	UF : 0, UT : 6,		CONFIG : 'N U T, 0, 0, 0',
	X =  520.535  mm,	Y =   -409.496  mm,	Z =   -242.091  mm,
	W =  90.000 deg,	P =   0.000 deg,	R =   90.000 deg
};
P[2300]{
   GP1:
	UF : 0, UT : 6,		CONFIG : 'N U T, 0, 0, 0',
	X =  519.132  mm,	Y =   -406.921  mm,	Z =   -241.887  mm,
	W =  90.000 deg,	P =   0.000 deg,	R =   90.000 deg
};
P[2301]{
   GP1:
	UF : 0, UT : 6,		CONFIG : 'N U T, 0, 0, 0',
	X =  518.741  mm,	Y =   -406.392  mm,	Z =   -242.094  mm,
	W =  90.000 deg,	P =   0.000 deg,	R =   90.000 deg
};
P[2302]{
   GP1:
	UF : 0, UT : 6,		CONFIG : 'N U T, 0, 0, 0',
	X =  518.272  mm,	Y =   -405.602  mm,	Z =   -242.126  mm,
	W =  90.000 deg,	P =   0.000 deg,	R =   90.000 deg
};
P[2303]{
   GP1:
	UF : 0, UT : 6,		CONFIG : 'N U T, 0, 0, 0',
	X =  517.990  mm,	Y =   -404.991  mm,	Z =   -241.953  mm,
	W =  90.000 deg,	P =   0.000 deg,	R =   90.000 deg
};
P[2304]{
   GP1:
	UF : 0, UT : 6,		CONFIG : 'N U T, 0, 0, 0',
	X =  516.646  mm,	Y =   -402.761  mm,	Z =   -242.092  mm,
	W =  90.000 deg,	P =   0.000 deg,	R =   90.000 deg
};
P[2305]{
   GP1:
	UF : 0, UT : 6,		CONFIG : 'N U T, 0, 0, 0',
	X =  515.812  mm,	Y =   -401.495  mm,	Z =   -242.341  mm,
	W =  90.000 deg,	P =   0.000 deg,	R =   90.000 deg
};
P[2306]{
   GP1:
	UF : 0, UT : 6,		CONFIG : 'N U T, 0, 0, 0',
	X =  515.649  mm,	Y =   -400.902  mm,	Z =   -241.904  mm,
	W =  90.000 deg,	P =   0.000 deg,	R =   90.000 deg
};
P[2307]{
   GP1:
	UF : 0, UT : 6,		CONFIG : 'N U T, 0, 0, 0',
	X =  513.969  mm,	Y =   -398.161  mm,	Z =   -242.142  mm,
	W =  90.000 deg,	P =   0.000 deg,	R =   90.000 deg
};
P[2308]{
   GP1:
	UF : 0, UT : 6,		CONFIG : 'N U T, 0, 0, 0',
	X =  513.252  mm,	Y =   -396.890  mm,	Z =   -242.102  mm,
	W =  90.000 deg,	P =   0.000 deg,	R =   90.000 deg
};
P[2309]{
   GP1:
	UF : 0, UT : 6,		CONFIG : 'N U T, 0, 0, 0',
	X =  511.571  mm,	Y =   -394.047  mm,	Z =   -242.197  mm,
	W =  90.000 deg,	P =   0.000 deg,	R =   90.000 deg
};
P[2310]{
   GP1:
	UF : 0, UT : 6,		CONFIG : 'N U T, 0, 0, 0',
	X =  511.208  mm,	Y =   -393.255  mm,	Z =   -241.967  mm,
	W =  90.000 deg,	P =   0.000 deg,	R =   90.000 deg
};
P[2311]{
   GP1:
	UF : 0, UT : 6,		CONFIG : 'N U T, 0, 0, 0',
	X =  510.489  mm,	Y =   -392.111  mm,	Z =   -242.110  mm,
	W =  90.000 deg,	P =   0.000 deg,	R =   90.000 deg
};
P[2312]{
   GP1:
	UF : 0, UT : 6,		CONFIG : 'N U T, 0, 0, 0',
	X =  509.945  mm,	Y =   -391.078  mm,	Z =   -241.984  mm,
	W =  90.000 deg,	P =   0.000 deg,	R =   90.000 deg
};
P[2313]{
   GP1:
	UF : 0, UT : 6,		CONFIG : 'N U T, 0, 0, 0',
	X =  508.918  mm,	Y =   -389.398  mm,	Z =   -242.119  mm,
	W =  90.000 deg,	P =   0.000 deg,	R =   90.000 deg
};
P[2314]{
   GP1:
	UF : 0, UT : 6,		CONFIG : 'N U T, 0, 0, 0',
	X =  507.426  mm,	Y =   -386.848  mm,	Z =   -242.167  mm,
	W =  90.000 deg,	P =   0.000 deg,	R =   90.000 deg
};
P[2315]{
   GP1:
	UF : 0, UT : 6,		CONFIG : 'N U T, 0, 0, 0',
	X =  506.566  mm,	Y =   -385.469  mm,	Z =   -242.323  mm,
	W =  90.000 deg,	P =   0.000 deg,	R =   90.000 deg
};
P[2316]{
   GP1:
	UF : 0, UT : 6,		CONFIG : 'N U T, 0, 0, 0',
	X =  504.503  mm,	Y =   -381.845  mm,	Z =   -242.253  mm,
	W =  90.000 deg,	P =   0.000 deg,	R =   90.000 deg
};
P[2317]{
   GP1:
	UF : 0, UT : 6,		CONFIG : 'N U T, 0, 0, 0',
	X =  503.831  mm,	Y =   -380.503  mm,	Z =   -242.002  mm,
	W =  90.000 deg,	P =   0.000 deg,	R =   90.000 deg
};
P[2318]{
   GP1:
	UF : 0, UT : 6,		CONFIG : 'N U T, 0, 0, 0',
	X =  503.104  mm,	Y =   -379.425  mm,	Z =   -242.256  mm,
	W =  90.000 deg,	P =   0.000 deg,	R =   90.000 deg
};
P[2319]{
   GP1:
	UF : 0, UT : 6,		CONFIG : 'N U T, 0, 0, 0',
	X =  502.548  mm,	Y =   -378.505  mm,	Z =   -242.316  mm,
	W =  90.000 deg,	P =   0.000 deg,	R =   90.000 deg
};
P[2320]{
   GP1:
	UF : 0, UT : 6,		CONFIG : 'N U T, 0, 0, 0',
	X =  501.117  mm,	Y =   -376.041  mm,	Z =   -242.337  mm,
	W =  90.000 deg,	P =   0.000 deg,	R =   90.000 deg
};
P[2321]{
   GP1:
	UF : 0, UT : 6,		CONFIG : 'N U T, 0, 0, 0',
	X =  500.740  mm,	Y =   -375.387  mm,	Z =   -242.336  mm,
	W =  90.000 deg,	P =   0.000 deg,	R =   90.000 deg
};
P[2322]{
   GP1:
	UF : 0, UT : 6,		CONFIG : 'N U T, 0, 0, 0',
	X =  498.713  mm,	Y =   -371.769  mm,	Z =   -242.182  mm,
	W =  90.000 deg,	P =   0.000 deg,	R =   90.000 deg
};
P[2323]{
   GP1:
	UF : 0, UT : 6,		CONFIG : 'N U T, 0, 0, 0',
	X =  497.056  mm,	Y =   -368.976  mm,	Z =   -242.291  mm,
	W =  90.000 deg,	P =   0.000 deg,	R =   90.000 deg
};
P[2324]{
   GP1:
	UF : 0, UT : 6,		CONFIG : 'N U T, 0, 0, 0',
	X =  495.655  mm,	Y =   -366.529  mm,	Z =   -242.264  mm,
	W =  90.000 deg,	P =   0.000 deg,	R =   90.000 deg
};
P[2325]{
   GP1:
	UF : 0, UT : 6,		CONFIG : 'N U T, 0, 0, 0',
	X =  495.105  mm,	Y =   -365.322  mm,	Z =   -241.906  mm,
	W =  90.000 deg,	P =   0.000 deg,	R =   90.000 deg
};
P[2326]{
   GP1:
	UF : 0, UT : 6,		CONFIG : 'N U T, 0, 0, 0',
	X =  493.399  mm,	Y =   -362.445  mm,	Z =   -242.015  mm,
	W =  90.000 deg,	P =   0.000 deg,	R =   90.000 deg
};
P[2327]{
   GP1:
	UF : 0, UT : 6,		CONFIG : 'N U T, 0, 0, 0',
	X =  492.705  mm,	Y =   -361.323  mm,	Z =   -242.125  mm,
	W =  90.000 deg,	P =   0.000 deg,	R =   90.000 deg
};
P[2328]{
   GP1:
	UF : 0, UT : 6,		CONFIG : 'N U T, 0, 0, 0',
	X =  490.298  mm,	Y =   -356.993  mm,	Z =   -241.900  mm,
	W =  90.000 deg,	P =   0.000 deg,	R =   90.000 deg
};
P[2329]{
   GP1:
	UF : 0, UT : 6,		CONFIG : 'N U T, 0, 0, 0',
	X =  489.670  mm,	Y =   -356.048  mm,	Z =   -242.102  mm,
	W =  90.000 deg,	P =   0.000 deg,	R =   90.000 deg
};
P[2330]{
   GP1:
	UF : 0, UT : 6,		CONFIG : 'N U T, 0, 0, 0',
	X =  489.326  mm,	Y =   -355.300  mm,	Z =   -241.887  mm,
	W =  90.000 deg,	P =   0.000 deg,	R =   90.000 deg
};
P[2331]{
   GP1:
	UF : 0, UT : 6,		CONFIG : 'N U T, 0, 0, 0',
	X =  486.930  mm,	Y =   -351.275  mm,	Z =   -242.063  mm,
	W =  90.000 deg,	P =   0.000 deg,	R =   90.000 deg
};
P[2332]{
   GP1:
	UF : 0, UT : 6,		CONFIG : 'N U T, 0, 0, 0',
	X =  486.384  mm,	Y =   -350.473  mm,	Z =   -242.263  mm,
	W =  90.000 deg,	P =   0.000 deg,	R =   90.000 deg
};
P[2333]{
   GP1:
	UF : 0, UT : 6,		CONFIG : 'N U T, 0, 0, 0',
	X =  484.114  mm,	Y =   -346.406  mm,	Z =   -242.074  mm,
	W =  90.000 deg,	P =   0.000 deg,	R =   90.000 deg
};
P[2334]{
   GP1:
	UF : 0, UT : 6,		CONFIG : 'N U T, 0, 0, 0',
	X =  483.617  mm,	Y =   -345.578  mm,	Z =   -242.119  mm,
	W =  90.000 deg,	P =   0.000 deg,	R =   90.000 deg
};
P[2335]{
   GP1:
	UF : 0, UT : 6,		CONFIG : 'N U T, 0, 0, 0',
	X =  482.584  mm,	Y =   -343.771  mm,	Z =   -242.094  mm,
	W =  90.000 deg,	P =   0.000 deg,	R =   90.000 deg
};
P[2336]{
   GP1:
	UF : 0, UT : 6,		CONFIG : 'N U T, 0, 0, 0',
	X =  481.565  mm,	Y =   -342.021  mm,	Z =   -242.115  mm,
	W =  90.000 deg,	P =   0.000 deg,	R =   90.000 deg
};
P[2337]{
   GP1:
	UF : 0, UT : 6,		CONFIG : 'N U T, 0, 0, 0',
	X =  479.797  mm,	Y =   -338.981  mm,	Z =   -242.147  mm,
	W =  90.000 deg,	P =   0.000 deg,	R =   90.000 deg
};
P[2338]{
   GP1:
	UF : 0, UT : 6,		CONFIG : 'N U T, 0, 0, 0',
	X =  479.119  mm,	Y =   -337.697  mm,	Z =   -241.992  mm,
	W =  90.000 deg,	P =   0.000 deg,	R =   90.000 deg
};
P[2339]{
   GP1:
	UF : 0, UT : 6,		CONFIG : 'N U T, 0, 0, 0',
	X =  478.316  mm,	Y =   -336.556  mm,	Z =   -242.343  mm,
	W =  90.000 deg,	P =   0.000 deg,	R =   90.000 deg
};
P[2340]{
   GP1:
	UF : 0, UT : 6,		CONFIG : 'N U T, 0, 0, 0',
	X =  477.952  mm,	Y =   -335.705  mm,	Z =   -242.033  mm,
	W =  90.000 deg,	P =   0.000 deg,	R =   90.000 deg
};
P[2341]{
   GP1:
	UF : 0, UT : 6,		CONFIG : 'N U T, 0, 0, 0',
	X =  476.685  mm,	Y =   -333.702  mm,	Z =   -242.302  mm,
	W =  90.000 deg,	P =   0.000 deg,	R =   90.000 deg
};
P[2342]{
   GP1:
	UF : 0, UT : 6,		CONFIG : 'N U T, 0, 0, 0',
	X =  476.046  mm,	Y =   -332.561  mm,	Z =   -242.253  mm,
	W =  90.000 deg,	P =   0.000 deg,	R =   90.000 deg
};
P[2343]{
   GP1:
	UF : 0, UT : 6,		CONFIG : 'N U T, 0, 0, 0',
	X =  475.573  mm,	Y =   -331.503  mm,	Z =   -241.919  mm,
	W =  90.000 deg,	P =   0.000 deg,	R =   90.000 deg
};
P[2344]{
   GP1:
	UF : 0, UT : 6,		CONFIG : 'N U T, 0, 0, 0',
	X =  474.795  mm,	Y =   -330.462  mm,	Z =   -242.346  mm,
	W =  90.000 deg,	P =   0.000 deg,	R =   90.000 deg
};
P[2345]{
   GP1:
	UF : 0, UT : 6,		CONFIG : 'N U T, 0, 0, 0',
	X =  474.193  mm,	Y =   -329.248  mm,	Z =   -242.106  mm,
	W =  90.000 deg,	P =   0.000 deg,	R =   90.000 deg
};
P[2346]{
   GP1:
	UF : 0, UT : 6,		CONFIG : 'N U T, 0, 0, 0',
	X =  473.672  mm,	Y =   -328.425  mm,	Z =   -242.218  mm,
	W =  90.000 deg,	P =   0.000 deg,	R =   90.000 deg
};
P[2347]{
   GP1:
	UF : 0, UT : 6,		CONFIG : 'N U T, 0, 0, 0',
	X =  472.228  mm,	Y =   -325.702  mm,	Z =   -241.909  mm,
	W =  90.000 deg,	P =   0.000 deg,	R =   90.000 deg
};
P[2348]{
   GP1:
	UF : 0, UT : 6,		CONFIG : 'N U T, 0, 0, 0',
	X =  470.347  mm,	Y =   -322.724  mm,	Z =   -242.299  mm,
	W =  90.000 deg,	P =   0.000 deg,	R =   90.000 deg
};
P[2349]{
   GP1:
	UF : 0, UT : 6,		CONFIG : 'N U T, 0, 0, 0',
	X =  469.866  mm,	Y =   -321.838  mm,	Z =   -242.225  mm,
	W =  90.000 deg,	P =   0.000 deg,	R =   90.000 deg
};
P[2350]{
   GP1:
	UF : 0, UT : 6,		CONFIG : 'N U T, 0, 0, 0',
	X =  468.693  mm,	Y =   -319.823  mm,	Z =   -242.249  mm,
	W =  90.000 deg,	P =   0.000 deg,	R =   90.000 deg
};
P[2351]{
   GP1:
	UF : 0, UT : 6,		CONFIG : 'N U T, 0, 0, 0',
	X =  467.380  mm,	Y =   -317.501  mm,	Z =   -242.183  mm,
	W =  90.000 deg,	P =   0.000 deg,	R =   90.000 deg
};
P[2352]{
   GP1:
	UF : 0, UT : 6,		CONFIG : 'N U T, 0, 0, 0',
	X =  463.139  mm,	Y =   -310.232  mm,	Z =   -242.290  mm,
	W =  90.000 deg,	P =   0.000 deg,	R =   90.000 deg
};
P[2353]{
   GP1:
	UF : 0, UT : 6,		CONFIG : 'N U T, 0, 0, 0',
	X =  461.944  mm,	Y =   -308.123  mm,	Z =   -242.234  mm,
	W =  90.000 deg,	P =   0.000 deg,	R =   90.000 deg
};
P[2354]{
   GP1:
	UF : 0, UT : 6,		CONFIG : 'N U T, 0, 0, 0',
	X =  459.569  mm,	Y =   -304.061  mm,	Z =   -242.304  mm,
	W =  90.000 deg,	P =   0.000 deg,	R =   90.000 deg
};
P[2355]{
   GP1:
	UF : 0, UT : 6,		CONFIG : 'N U T, 0, 0, 0',
	X =  458.242  mm,	Y =   -301.713  mm,	Z =   -242.237  mm,
	W =  90.000 deg,	P =   0.000 deg,	R =   90.000 deg
};
P[2356]{
   GP1:
	UF : 0, UT : 6,		CONFIG : 'N U T, 0, 0, 0',
	X =  457.767  mm,	Y =   -300.851  mm,	Z =   -242.180  mm,
	W =  90.000 deg,	P =   0.000 deg,	R =   90.000 deg
};
P[2357]{
   GP1:
	UF : 0, UT : 6,		CONFIG : 'N U T, 0, 0, 0',
	X =  456.514  mm,	Y =   -298.800  mm,	Z =   -242.345  mm,
	W =  90.000 deg,	P =   0.000 deg,	R =   90.000 deg
};
P[2358]{
   GP1:
	UF : 0, UT : 6,		CONFIG : 'N U T, 0, 0, 0',
	X =  455.452  mm,	Y =   -296.841  mm,	Z =   -242.180  mm,
	W =  90.000 deg,	P =   0.000 deg,	R =   90.000 deg
};
P[2359]{
   GP1:
	UF : 0, UT : 6,		CONFIG : 'N U T, 0, 0, 0',
	X =  453.945  mm,	Y =   -294.284  mm,	Z =   -242.252  mm,
	W =  90.000 deg,	P =   0.000 deg,	R =   90.000 deg
};
P[2360]{
   GP1:
	UF : 0, UT : 6,		CONFIG : 'N U T, 0, 0, 0',
	X =  453.336  mm,	Y =   -293.191  mm,	Z =   -242.200  mm,
	W =  90.000 deg,	P =   0.000 deg,	R =   90.000 deg
};
P[2361]{
   GP1:
	UF : 0, UT : 6,		CONFIG : 'N U T, 0, 0, 0',
	X =  451.909  mm,	Y =   -290.780  mm,	Z =   -242.285  mm,
	W =  90.000 deg,	P =   0.000 deg,	R =   90.000 deg
};
P[2362]{
   GP1:
	UF : 0, UT : 6,		CONFIG : 'N U T, 0, 0, 0',
	X =  451.301  mm,	Y =   -289.602  mm,	Z =   -242.110  mm,
	W =  90.000 deg,	P =   0.000 deg,	R =   90.000 deg
};
P[2363]{
   GP1:
	UF : 0, UT : 6,		CONFIG : 'N U T, 0, 0, 0',
	X =  450.675  mm,	Y =   -288.637  mm,	Z =   -242.277  mm,
	W =  90.000 deg,	P =   0.000 deg,	R =   90.000 deg
};
P[2364]{
   GP1:
	UF : 0, UT : 6,		CONFIG : 'N U T, 0, 0, 0',
	X =  447.511  mm,	Y =   -282.907  mm,	Z =   -241.926  mm,
	W =  90.000 deg,	P =   0.000 deg,	R =   90.000 deg
};
P[2365]{
   GP1:
	UF : 0, UT : 6,		CONFIG : 'N U T, 0, 0, 0',
	X =  446.673  mm,	Y =   -281.438  mm,	Z =   -241.901  mm,
	W =  90.000 deg,	P =   0.000 deg,	R =   90.000 deg
};
P[2366]{
   GP1:
	UF : 0, UT : 6,		CONFIG : 'N U T, 0, 0, 0',
	X =  446.075  mm,	Y =   -280.671  mm,	Z =   -242.278  mm,
	W =  90.000 deg,	P =   0.000 deg,	R =   90.000 deg
};
P[2367]{
   GP1:
	UF : 0, UT : 6,		CONFIG : 'N U T, 0, 0, 0',
	X =  445.596  mm,	Y =   -279.837  mm,	Z =   -242.272  mm,
	W =  90.000 deg,	P =   0.000 deg,	R =   90.000 deg
};
P[2368]{
   GP1:
	UF : 0, UT : 6,		CONFIG : 'N U T, 0, 0, 0',
	X =  444.248  mm,	Y =   -277.232  mm,	Z =   -241.892  mm,
	W =  90.000 deg,	P =   0.000 deg,	R =   90.000 deg
};
P[2369]{
   GP1:
	UF : 0, UT : 6,		CONFIG : 'N U T, 0, 0, 0',
	X =  443.694  mm,	Y =   -276.618  mm,	Z =   -242.375  mm,
	W =  90.000 deg,	P =   0.000 deg,	R =   90.000 deg
};
P[2370]{
   GP1:
	UF : 0, UT : 6,		CONFIG : 'N U T, 0, 0, 0',
	X =  443.562  mm,	Y =   -276.084  mm,	Z =   -241.947  mm,
	W =  90.000 deg,	P =   0.000 deg,	R =   90.000 deg
};
P[2371]{
   GP1:
	UF : 0, UT : 6,		CONFIG : 'N U T, 0, 0, 0',
	X =  441.368  mm,	Y =   -272.447  mm,	Z =   -242.179  mm,
	W =  90.000 deg,	P =   0.000 deg,	R =   90.000 deg
};
P[2372]{
   GP1:
	UF : 0, UT : 6,		CONFIG : 'N U T, 0, 0, 0',
	X =  440.822  mm,	Y =   -271.628  mm,	Z =   -242.353  mm,
	W =  90.000 deg,	P =   0.000 deg,	R =   90.000 deg
};
P[2373]{
   GP1:
	UF : 0, UT : 6,		CONFIG : 'N U T, 0, 0, 0',
	X =  440.496  mm,	Y =   -270.871  mm,	Z =   -242.085  mm,
	W =  90.000 deg,	P =   0.000 deg,	R =   90.000 deg
};
P[2374]{
   GP1:
	UF : 0, UT : 6,		CONFIG : 'N U T, 0, 0, 0',
	X =  439.962  mm,	Y =   -270.155  mm,	Z =   -242.379  mm,
	W =  90.000 deg,	P =   0.000 deg,	R =   90.000 deg
};
P[2375]{
   GP1:
	UF : 0, UT : 6,		CONFIG : 'N U T, 0, 0, 0',
	X =  437.041  mm,	Y =   -264.977  mm,	Z =   -242.210  mm,
	W =  90.000 deg,	P =   0.000 deg,	R =   90.000 deg
};
P[2376]{
   GP1:
	UF : 0, UT : 6,		CONFIG : 'N U T, 0, 0, 0',
	X =  436.366  mm,	Y =   -263.921  mm,	Z =   -242.372  mm,
	W =  90.000 deg,	P =   0.000 deg,	R =   90.000 deg
};
P[2377]{
   GP1:
	UF : 0, UT : 6,		CONFIG : 'N U T, 0, 0, 0',
	X =  435.930  mm,	Y =   -263.107  mm,	Z =   -242.285  mm,
	W =  90.000 deg,	P =   0.000 deg,	R =   90.000 deg
};
P[2378]{
   GP1:
	UF : 0, UT : 6,		CONFIG : 'N U T, 0, 0, 0',
	X =  435.253  mm,	Y =   -261.728  mm,	Z =   -241.997  mm,
	W =  90.000 deg,	P =   0.000 deg,	R =   90.000 deg
};
P[2379]{
   GP1:
	UF : 0, UT : 6,		CONFIG : 'N U T, 0, 0, 0',
	X =  433.995  mm,	Y =   -259.677  mm,	Z =   -242.175  mm,
	W =  90.000 deg,	P =   0.000 deg,	R =   90.000 deg
};
P[2380]{
   GP1:
	UF : 0, UT : 6,		CONFIG : 'N U T, 0, 0, 0',
	X =  432.424  mm,	Y =   -256.757  mm,	Z =   -241.899  mm,
	W =  90.000 deg,	P =   0.000 deg,	R =   90.000 deg
};
P[2381]{
   GP1:
	UF : 0, UT : 6,		CONFIG : 'N U T, 0, 0, 0',
	X =  429.671  mm,	Y =   -252.047  mm,	Z =   -241.978  mm,
	W =  90.000 deg,	P =   0.000 deg,	R =   90.000 deg
};
P[2382]{
   GP1:
	UF : 0, UT : 6,		CONFIG : 'N U T, 0, 0, 0',
	X =  428.849  mm,	Y =   -250.891  mm,	Z =   -242.353  mm,
	W =  90.000 deg,	P =   0.000 deg,	R =   90.000 deg
};
P[2383]{
   GP1:
	UF : 0, UT : 6,		CONFIG : 'N U T, 0, 0, 0',
	X =  428.198  mm,	Y =   -249.636  mm,	Z =   -242.174  mm,
	W =  90.000 deg,	P =   0.000 deg,	R =   90.000 deg
};
P[2384]{
   GP1:
	UF : 0, UT : 6,		CONFIG : 'N U T, 0, 0, 0',
	X =  426.373  mm,	Y =   -246.561  mm,	Z =   -242.295  mm,
	W =  90.000 deg,	P =   0.000 deg,	R =   90.000 deg
};
P[2385]{
   GP1:
	UF : 0, UT : 6,		CONFIG : 'N U T, 0, 0, 0',
	X =  425.315  mm,	Y =   -244.465  mm,	Z =   -241.925  mm,
	W =  90.000 deg,	P =   0.000 deg,	R =   90.000 deg
};
P[2386]{
   GP1:
	UF : 0, UT : 6,		CONFIG : 'N U T, 0, 0, 0',
	X =  424.413  mm,	Y =   -243.120  mm,	Z =   -242.231  mm,
	W =  90.000 deg,	P =   0.000 deg,	R =   90.000 deg
};
P[2387]{
   GP1:
	UF : 0, UT : 6,		CONFIG : 'N U T, 0, 0, 0',
	X =  423.533  mm,	Y =   -241.506  mm,	Z =   -242.105  mm,
	W =  90.000 deg,	P =   0.000 deg,	R =   90.000 deg
};
P[2388]{
   GP1:
	UF : 0, UT : 6,		CONFIG : 'N U T, 0, 0, 0',
	X =  422.236  mm,	Y =   -239.270  mm,	Z =   -242.117  mm,
	W =  90.000 deg,	P =   0.000 deg,	R =   90.000 deg
};
P[2389]{
   GP1:
	UF : 0, UT : 6,		CONFIG : 'N U T, 0, 0, 0',
	X =  419.654  mm,	Y =   -234.838  mm,	Z =   -242.176  mm,
	W =  90.000 deg,	P =   0.000 deg,	R =   90.000 deg
};
P[2390]{
   GP1:
	UF : 0, UT : 6,		CONFIG : 'N U T, 0, 0, 0',
	X =  418.527  mm,	Y =   -232.974  mm,	Z =   -242.298  mm,
	W =  90.000 deg,	P =   0.000 deg,	R =   90.000 deg
};
P[2391]{
   GP1:
	UF : 0, UT : 6,		CONFIG : 'N U T, 0, 0, 0',
	X =  418.182  mm,	Y =   -232.092  mm,	Z =   -241.898  mm,
	W =  90.000 deg,	P =   0.000 deg,	R =   90.000 deg
};
P[2392]{
   GP1:
	UF : 0, UT : 6,		CONFIG : 'N U T, 0, 0, 0',
	X =  416.419  mm,	Y =   -229.347  mm,	Z =   -242.330  mm,
	W =  90.000 deg,	P =   0.000 deg,	R =   90.000 deg
};
P[2393]{
   GP1:
	UF : 0, UT : 6,		CONFIG : 'N U T, 0, 0, 0',
	X =  413.412  mm,	Y =   -224.010  mm,	Z =   -242.151  mm,
	W =  90.000 deg,	P =   0.000 deg,	R =   90.000 deg
};
P[2394]{
   GP1:
	UF : 0, UT : 6,		CONFIG : 'N U T, 0, 0, 0',
	X =  411.302  mm,	Y =   -220.419  mm,	Z =   -242.240  mm,
	W =  90.000 deg,	P =   0.000 deg,	R =   90.000 deg
};
P[2395]{
   GP1:
	UF : 0, UT : 6,		CONFIG : 'N U T, 0, 0, 0',
	X =  410.712  mm,	Y =   -219.255  mm,	Z =   -242.040  mm,
	W =  90.000 deg,	P =   0.000 deg,	R =   90.000 deg
};
P[2396]{
   GP1:
	UF : 0, UT : 6,		CONFIG : 'N U T, 0, 0, 0',
	X =  410.074  mm,	Y =   -218.268  mm,	Z =   -242.206  mm,
	W =  90.000 deg,	P =   0.000 deg,	R =   90.000 deg
};
P[2397]{
   GP1:
	UF : 0, UT : 6,		CONFIG : 'N U T, 0, 0, 0',
	X =  409.057  mm,	Y =   -216.460  mm,	Z =   -242.140  mm,
	W =  90.000 deg,	P =   0.000 deg,	R =   90.000 deg
};
P[2398]{
   GP1:
	UF : 0, UT : 6,		CONFIG : 'N U T, 0, 0, 0',
	X =  407.877  mm,	Y =   -214.526  mm,	Z =   -242.295  mm,
	W =  90.000 deg,	P =   0.000 deg,	R =   90.000 deg
};
P[2399]{
   GP1:
	UF : 0, UT : 6,		CONFIG : 'N U T, 0, 0, 0',
	X =  406.464  mm,	Y =   -211.948  mm,	Z =   -242.110  mm,
	W =  90.000 deg,	P =   0.000 deg,	R =   90.000 deg
};
P[2400]{
   GP1:
	UF : 0, UT : 6,		CONFIG : 'N U T, 0, 0, 0',
	X =  404.906  mm,	Y =   -209.428  mm,	Z =   -242.361  mm,
	W =  90.000 deg,	P =   0.000 deg,	R =   90.000 deg
};
P[2401]{
   GP1:
	UF : 0, UT : 6,		CONFIG : 'N U T, 0, 0, 0',
	X =  403.982  mm,	Y =   -207.625  mm,	Z =   -242.075  mm,
	W =  90.000 deg,	P =   0.000 deg,	R =   90.000 deg
};
P[2402]{
   GP1:
	UF : 0, UT : 6,		CONFIG : 'N U T, 0, 0, 0',
	X =  398.838  mm,	Y =   -198.889  mm,	Z =   -242.318  mm,
	W =  90.000 deg,	P =   0.000 deg,	R =   90.000 deg
};
P[2403]{
   GP1:
	UF : 0, UT : 6,		CONFIG : 'N U T, 0, 0, 0',
	X =  397.944  mm,	Y =   -197.338  mm,	Z =   -242.313  mm,
	W =  90.000 deg,	P =   0.000 deg,	R =   90.000 deg
};
P[2404]{
   GP1:
	UF : 0, UT : 6,		CONFIG : 'N U T, 0, 0, 0',
	X =  396.427  mm,	Y =   -194.589  mm,	Z =   -242.145  mm,
	W =  90.000 deg,	P =   0.000 deg,	R =   90.000 deg
};
P[2405]{
   GP1:
	UF : 0, UT : 6,		CONFIG : 'N U T, 0, 0, 0',
	X =  395.866  mm,	Y =   -193.571  mm,	Z =   -242.078  mm,
	W =  90.000 deg,	P =   0.000 deg,	R =   90.000 deg
};
P[2406]{
   GP1:
	UF : 0, UT : 6,		CONFIG : 'N U T, 0, 0, 0',
	X =  394.828  mm,	Y =   -191.769  mm,	Z =   -242.075  mm,
	W =  90.000 deg,	P =   0.000 deg,	R =   90.000 deg
};
P[2407]{
   GP1:
	UF : 0, UT : 6,		CONFIG : 'N U T, 0, 0, 0',
	X =  392.816  mm,	Y =   -188.213  mm,	Z =   -241.973  mm,
	W =  90.000 deg,	P =   0.000 deg,	R =   90.000 deg
};
P[2408]{
   GP1:
	UF : 0, UT : 6,		CONFIG : 'N U T, 0, 0, 0',
	X =  389.657  mm,	Y =   -182.872  mm,	Z =   -242.158  mm,
	W =  90.000 deg,	P =   0.000 deg,	R =   90.000 deg
};
P[2409]{
   GP1:
	UF : 0, UT : 6,		CONFIG : 'N U T, 0, 0, 0',
	X =  388.707  mm,	Y =   -181.037  mm,	Z =   -241.889  mm,
	W =  90.000 deg,	P =   0.000 deg,	R =   90.000 deg
};
P[2410]{
   GP1:
	UF : 0, UT : 6,		CONFIG : 'N U T, 0, 0, 0',
	X =  387.311  mm,	Y =   -178.764  mm,	Z =   -242.095  mm,
	W =  90.000 deg,	P =   0.000 deg,	R =   90.000 deg
};
P[2411]{
   GP1:
	UF : 0, UT : 6,		CONFIG : 'N U T, 0, 0, 0',
	X =  384.702  mm,	Y =   -174.381  mm,	Z =   -242.282  mm,
	W =  90.000 deg,	P =   0.000 deg,	R =   90.000 deg
};
P[2412]{
   GP1:
	UF : 0, UT : 6,		CONFIG : 'N U T, 0, 0, 0',
	X =  384.296  mm,	Y =   -173.622  mm,	Z =   -242.207  mm,
	W =  90.000 deg,	P =   0.000 deg,	R =   90.000 deg
};
P[2413]{
   GP1:
	UF : 0, UT : 6,		CONFIG : 'N U T, 0, 0, 0',
	X =  383.752  mm,	Y =   -172.767  mm,	Z =   -242.326  mm,
	W =  90.000 deg,	P =   0.000 deg,	R =   90.000 deg
};
P[2414]{
   GP1:
	UF : 0, UT : 6,		CONFIG : 'N U T, 0, 0, 0',
	X =  380.866  mm,	Y =   -167.749  mm,	Z =   -242.300  mm,
	W =  90.000 deg,	P =   0.000 deg,	R =   90.000 deg
};
P[2415]{
   GP1:
	UF : 0, UT : 6,		CONFIG : 'N U T, 0, 0, 0',
	X =  377.409  mm,	Y =   -161.701  mm,	Z =   -242.214  mm,
	W =  90.000 deg,	P =   0.000 deg,	R =   90.000 deg
};
P[2416]{
   GP1:
	UF : 0, UT : 6,		CONFIG : 'N U T, 0, 0, 0',
	X =  374.971  mm,	Y =   -157.493  mm,	Z =   -242.236  mm,
	W =  90.000 deg,	P =   0.000 deg,	R =   90.000 deg
};
P[2417]{
   GP1:
	UF : 0, UT : 6,		CONFIG : 'N U T, 0, 0, 0',
	X =  373.275  mm,	Y =   -154.514  mm,	Z =   -242.176  mm,
	W =  90.000 deg,	P =   0.000 deg,	R =   90.000 deg
};
P[2418]{
   GP1:
	UF : 0, UT : 6,		CONFIG : 'N U T, 0, 0, 0',
	X =  372.493  mm,	Y =   -152.966  mm,	Z =   -241.903  mm,
	W =  90.000 deg,	P =   0.000 deg,	R =   90.000 deg
};
P[2419]{
   GP1:
	UF : 0, UT : 6,		CONFIG : 'N U T, 0, 0, 0',
	X =  371.671  mm,	Y =   -151.834  mm,	Z =   -242.312  mm,
	W =  90.000 deg,	P =   0.000 deg,	R =   90.000 deg
};
P[2420]{
   GP1:
	UF : 0, UT : 6,		CONFIG : 'N U T, 0, 0, 0',
	X =  371.217  mm,	Y =   -151.067  mm,	Z =   -242.340  mm,
	W =  90.000 deg,	P =   0.000 deg,	R =   90.000 deg
};
P[2421]{
   GP1:
	UF : 0, UT : 6,		CONFIG : 'N U T, 0, 0, 0',
	X =  370.776  mm,	Y =   -150.185  mm,	Z =   -242.177  mm,
	W =  90.000 deg,	P =   0.000 deg,	R =   90.000 deg
};
P[2422]{
   GP1:
	UF : 0, UT : 6,		CONFIG : 'N U T, 0, 0, 0',
	X =  369.503  mm,	Y =   -148.020  mm,	Z =   -242.230  mm,
	W =  90.000 deg,	P =   0.000 deg,	R =   90.000 deg
};
P[2423]{
   GP1:
	UF : 0, UT : 6,		CONFIG : 'N U T, 0, 0, 0',
	X =  368.638  mm,	Y =   -146.346  mm,	Z =   -241.985  mm,
	W =  90.000 deg,	P =   0.000 deg,	R =   90.000 deg
};
P[2424]{
   GP1:
	UF : 0, UT : 6,		CONFIG : 'N U T, 0, 0, 0',
	X =  366.205  mm,	Y =   -142.407  mm,	Z =   -242.371  mm,
	W =  90.000 deg,	P =   0.000 deg,	R =   90.000 deg
};
P[2425]{
   GP1:
	UF : 0, UT : 6,		CONFIG : 'N U T, 0, 0, 0',
	X =  365.745  mm,	Y =   -141.523  mm,	Z =   -242.246  mm,
	W =  90.000 deg,	P =   0.000 deg,	R =   90.000 deg
};
P[2426]{
   GP1:
	UF : 0, UT : 6,		CONFIG : 'N U T, 0, 0, 0',
	X =  364.150  mm,	Y =   -138.854  mm,	Z =   -242.379  mm,
	W =  90.000 deg,	P =   0.000 deg,	R =   90.000 deg
};
P[2427]{
   GP1:
	UF : 0, UT : 6,		CONFIG : 'N U T, 0, 0, 0',
	X =  361.279  mm,	Y =   -133.867  mm,	Z =   -242.358  mm,
	W =  90.000 deg,	P =   0.000 deg,	R =   90.000 deg
};
P[2428]{
   GP1:
	UF : 0, UT : 6,		CONFIG : 'N U T, 0, 0, 0',
	X =  360.164  mm,	Y =   -131.751  mm,	Z =   -242.100  mm,
	W =  90.000 deg,	P =   0.000 deg,	R =   90.000 deg
};
P[2429]{
   GP1:
	UF : 0, UT : 6,		CONFIG : 'N U T, 0, 0, 0',
	X =  359.741  mm,	Y =   -130.894  mm,	Z =   -241.924  mm,
	W =  90.000 deg,	P =   0.000 deg,	R =   90.000 deg
};
P[2430]{
   GP1:
	UF : 0, UT : 6,		CONFIG : 'N U T, 0, 0, 0',
	X =  359.264  mm,	Y =   -130.362  mm,	Z =   -242.336  mm,
	W =  90.000 deg,	P =   0.000 deg,	R =   90.000 deg
};
P[2431]{
   GP1:
	UF : 0, UT : 6,		CONFIG : 'N U T, 0, 0, 0',
	X =  358.767  mm,	Y =   -129.206  mm,	Z =   -241.925  mm,
	W =  90.000 deg,	P =   0.000 deg,	R =   90.000 deg
};
P[2432]{
   GP1:
	UF : 0, UT : 6,		CONFIG : 'N U T, 0, 0, 0',
	X =  356.711  mm,	Y =   -125.784  mm,	Z =   -242.118  mm,
	W =  90.000 deg,	P =   0.000 deg,	R =   90.000 deg
};
P[2433]{
   GP1:
	UF : 0, UT : 6,		CONFIG : 'N U T, 0, 0, 0',
	X =  355.868  mm,	Y =   -124.513  mm,	Z =   -242.381  mm,
	W =  90.000 deg,	P =   0.000 deg,	R =   90.000 deg
};
P[2434]{
   GP1:
	UF : 0, UT : 6,		CONFIG : 'N U T, 0, 0, 0',
	X =  353.188  mm,	Y =   -119.945  mm,	Z =   -242.066  mm,
	W =  90.000 deg,	P =   0.000 deg,	R =   90.000 deg
};
P[2435]{
   GP1:
	UF : 0, UT : 6,		CONFIG : 'N U T, 0, 0, 0',
	X =  351.575  mm,	Y =   -117.960  mm,	Z =   -241.889  mm,
	W =  90.000 deg,	P =   0.000 deg,	R =   90.000 deg
};
P[2436]{
   GP1:
	UF : 0, UT : 6,		CONFIG : 'N U T, 0, 0, 0',
	X =  350.981  mm,	Y =   -117.434  mm,	Z =   -241.919  mm,
	W =  90.000 deg,	P =   0.000 deg,	R =   90.000 deg
};
P[2437]{
   GP1:
	UF : 0, UT : 6,		CONFIG : 'N U T, 0, 0, 0',
	X =  349.938  mm,	Y =   -116.796  mm,	Z =   -242.267  mm,
	W =  90.000 deg,	P =   0.000 deg,	R =   90.000 deg
};
P[2438]{
   GP1:
	UF : 0, UT : 6,		CONFIG : 'N U T, 0, 0, 0',
	X =  348.991  mm,	Y =   -116.126  mm,	Z =   -242.123  mm,
	W =  90.000 deg,	P =   0.000 deg,	R =   90.000 deg
};
P[2439]{
   GP1:
	UF : 0, UT : 6,		CONFIG : 'N U T, 0, 0, 0',
	X =  347.743  mm,	Y =   -115.542  mm,	Z =   -242.284  mm,
	W =  90.000 deg,	P =   0.000 deg,	R =   90.000 deg
};
P[2440]{
   GP1:
	UF : 0, UT : 6,		CONFIG : 'N U T, 0, 0, 0',
	X =  344.288  mm,	Y =   -114.583  mm,	Z =   -242.382  mm,
	W =  90.000 deg,	P =   0.000 deg,	R =   90.000 deg
};
P[2441]{
   GP1:
	UF : 0, UT : 6,		CONFIG : 'N U T, 0, 0, 0',
	X =  343.306  mm,	Y =   -114.342  mm,	Z =   -242.136  mm,
	W =  90.000 deg,	P =   0.000 deg,	R =   90.000 deg
};
P[2442]{
   GP1:
	UF : 0, UT : 6,		CONFIG : 'N U T, 0, 0, 0',
	X =  342.224  mm,	Y =   -114.391  mm,	Z =   -242.272  mm,
	W =  90.000 deg,	P =   0.000 deg,	R =   90.000 deg
};
P[2443]{
   GP1:
	UF : 0, UT : 6,		CONFIG : 'N U T, 0, 0, 0',
	X =  340.298  mm,	Y =   -114.527  mm,	Z =   -242.266  mm,
	W =  90.000 deg,	P =   0.000 deg,	R =   90.000 deg
};
P[2444]{
   GP1:
	UF : 0, UT : 6,		CONFIG : 'N U T, 0, 0, 0',
	X =  337.448  mm,	Y =   -115.270  mm,	Z =   -242.255  mm,
	W =  90.000 deg,	P =   0.000 deg,	R =   90.000 deg
};
P[2445]{
   GP1:
	UF : 0, UT : 6,		CONFIG : 'N U T, 0, 0, 0',
	X =  336.767  mm,	Y =   -115.426  mm,	Z =   -241.918  mm,
	W =  90.000 deg,	P =   0.000 deg,	R =   90.000 deg
};
P[2446]{
   GP1:
	UF : 0, UT : 6,		CONFIG : 'N U T, 0, 0, 0',
	X =  335.548  mm,	Y =   -116.136  mm,	Z =   -242.263  mm,
	W =  90.000 deg,	P =   0.000 deg,	R =   90.000 deg
};
P[2447]{
   GP1:
	UF : 0, UT : 6,		CONFIG : 'N U T, 0, 0, 0',
	X =  333.946  mm,	Y =   -116.937  mm,	Z =   -242.070  mm,
	W =  90.000 deg,	P =   0.000 deg,	R =   90.000 deg
};
P[2448]{
   GP1:
	UF : 0, UT : 6,		CONFIG : 'N U T, 0, 0, 0',
	X =  332.979  mm,	Y =   -117.584  mm,	Z =   -242.281  mm,
	W =  90.000 deg,	P =   0.000 deg,	R =   90.000 deg
};
P[2449]{
   GP1:
	UF : 0, UT : 6,		CONFIG : 'N U T, 0, 0, 0',
	X =  330.242  mm,	Y =   -119.206  mm,	Z =   -242.385  mm,
	W =  90.000 deg,	P =   0.000 deg,	R =   90.000 deg
};
P[2450]{
   GP1:
	UF : 0, UT : 6,		CONFIG : 'N U T, 0, 0, 0',
	X =  325.927  mm,	Y =   -121.586  mm,	Z =   -242.114  mm,
	W =  90.000 deg,	P =   0.000 deg,	R =   90.000 deg
};
P[2451]{
   GP1:
	UF : 0, UT : 6,		CONFIG : 'N U T, 0, 0, 0',
	X =  325.100  mm,	Y =   -122.063  mm,	Z =   -242.114  mm,
	W =  90.000 deg,	P =   0.000 deg,	R =   90.000 deg
};
P[2452]{
   GP1:
	UF : 0, UT : 6,		CONFIG : 'N U T, 0, 0, 0',
	X =  321.438  mm,	Y =   -124.140  mm,	Z =   -242.024  mm,
	W =  90.000 deg,	P =   0.000 deg,	R =   90.000 deg
};
P[2453]{
   GP1:
	UF : 0, UT : 6,		CONFIG : 'N U T, 0, 0, 0',
	X =  318.802  mm,	Y =   -125.797  mm,	Z =   -242.348  mm,
	W =  90.000 deg,	P =   0.000 deg,	R =   90.000 deg
};
P[2454]{
   GP1:
	UF : 0, UT : 6,		CONFIG : 'N U T, 0, 0, 0',
	X =  315.382  mm,	Y =   -127.677  mm,	Z =   -242.119  mm,
	W =  90.000 deg,	P =   0.000 deg,	R =   90.000 deg
};
P[2455]{
   GP1:
	UF : 0, UT : 6,		CONFIG : 'N U T, 0, 0, 0',
	X =  314.044  mm,	Y =   -128.543  mm,	Z =   -242.346  mm,
	W =  90.000 deg,	P =   0.000 deg,	R =   90.000 deg
};
P[2456]{
   GP1:
	UF : 0, UT : 6,		CONFIG : 'N U T, 0, 0, 0',
	X =  313.417  mm,	Y =   -128.917  mm,	Z =   -242.376  mm,
	W =  90.000 deg,	P =   0.000 deg,	R =   90.000 deg
};
P[2457]{
   GP1:
	UF : 0, UT : 6,		CONFIG : 'N U T, 0, 0, 0',
	X =  310.933  mm,	Y =   -130.286  mm,	Z =   -242.216  mm,
	W =  90.000 deg,	P =   0.000 deg,	R =   90.000 deg
};
P[2458]{
   GP1:
	UF : 0, UT : 6,		CONFIG : 'N U T, 0, 0, 0',
	X =  309.377  mm,	Y =   -131.142  mm,	Z =   -242.112  mm,
	W =  90.000 deg,	P =   0.000 deg,	R =   90.000 deg
};
P[2459]{
   GP1:
	UF : 0, UT : 6,		CONFIG : 'N U T, 0, 0, 0',
	X =  306.926  mm,	Y =   -132.473  mm,	Z =   -241.910  mm,
	W =  90.000 deg,	P =   0.000 deg,	R =   90.000 deg
};
P[2460]{
   GP1:
	UF : 0, UT : 6,		CONFIG : 'N U T, 0, 0, 0',
	X =  300.411  mm,	Y =   -136.322  mm,	Z =   -242.120  mm,
	W =  90.000 deg,	P =   0.000 deg,	R =   90.000 deg
};
P[2461]{
   GP1:
	UF : 0, UT : 6,		CONFIG : 'N U T, 0, 0, 0',
	X =  299.845  mm,	Y =   -136.737  mm,	Z =   -242.335  mm,
	W =  90.000 deg,	P =   0.000 deg,	R =   90.000 deg
};
P[2462]{
   GP1:
	UF : 0, UT : 6,		CONFIG : 'N U T, 0, 0, 0',
	X =  297.738  mm,	Y =   -137.880  mm,	Z =   -242.156  mm,
	W =  90.000 deg,	P =   0.000 deg,	R =   90.000 deg
};
P[2463]{
   GP1:
	UF : 0, UT : 6,		CONFIG : 'N U T, 0, 0, 0',
	X =  295.999  mm,	Y =   -138.813  mm,	Z =   -241.983  mm,
	W =  90.000 deg,	P =   0.000 deg,	R =   90.000 deg
};
P[2464]{
   GP1:
	UF : 0, UT : 6,		CONFIG : 'N U T, 0, 0, 0',
	X =  294.607  mm,	Y =   -139.699  mm,	Z =   -242.185  mm,
	W =  90.000 deg,	P =   0.000 deg,	R =   90.000 deg
};
P[2465]{
   GP1:
	UF : 0, UT : 6,		CONFIG : 'N U T, 0, 0, 0',
	X =  291.787  mm,	Y =   -141.316  mm,	Z =   -242.156  mm,
	W =  90.000 deg,	P =   0.000 deg,	R =   90.000 deg
};
P[2466]{
   GP1:
	UF : 0, UT : 6,		CONFIG : 'N U T, 0, 0, 0',
	X =  289.540  mm,	Y =   -142.637  mm,	Z =   -242.214  mm,
	W =  90.000 deg,	P =   0.000 deg,	R =   90.000 deg
};
P[2467]{
   GP1:
	UF : 0, UT : 6,		CONFIG : 'N U T, 0, 0, 0',
	X =  286.156  mm,	Y =   -144.572  mm,	Z =   -242.167  mm,
	W =  90.000 deg,	P =   0.000 deg,	R =   90.000 deg
};
P[2468]{
   GP1:
	UF : 0, UT : 6,		CONFIG : 'N U T, 0, 0, 0',
	X =  282.733  mm,	Y =   -146.447  mm,	Z =   -241.919  mm,
	W =  90.000 deg,	P =   0.000 deg,	R =   90.000 deg
};
P[2469]{
   GP1:
	UF : 0, UT : 6,		CONFIG : 'N U T, 0, 0, 0',
	X =  282.110  mm,	Y =   -146.948  mm,	Z =   -242.266  mm,
	W =  90.000 deg,	P =   0.000 deg,	R =   90.000 deg
};
P[2470]{
   GP1:
	UF : 0, UT : 6,		CONFIG : 'N U T, 0, 0, 0',
	X =  281.219  mm,	Y =   -147.479  mm,	Z =   -242.303  mm,
	W =  90.000 deg,	P =   0.000 deg,	R =   90.000 deg
};
P[2471]{
   GP1:
	UF : 0, UT : 6,		CONFIG : 'N U T, 0, 0, 0',
	X =  280.131  mm,	Y =   -148.009  mm,	Z =   -242.066  mm,
	W =  90.000 deg,	P =   0.000 deg,	R =   90.000 deg
};
P[2472]{
   GP1:
	UF : 0, UT : 6,		CONFIG : 'N U T, 0, 0, 0',
	X =  278.798  mm,	Y =   -148.793  mm,	Z =   -242.100  mm,
	W =  90.000 deg,	P =   0.000 deg,	R =   90.000 deg
};
P[2473]{
   GP1:
	UF : 0, UT : 6,		CONFIG : 'N U T, 0, 0, 0',
	X =  277.780  mm,	Y =   -149.353  mm,	Z =   -242.033  mm,
	W =  90.000 deg,	P =   0.000 deg,	R =   90.000 deg
};
P[2474]{
   GP1:
	UF : 0, UT : 6,		CONFIG : 'N U T, 0, 0, 0',
	X =  276.966  mm,	Y =   -149.917  mm,	Z =   -242.260  mm,
	W =  90.000 deg,	P =   0.000 deg,	R =   90.000 deg
};
P[2475]{
   GP1:
	UF : 0, UT : 6,		CONFIG : 'N U T, 0, 0, 0',
	X =  274.377  mm,	Y =   -151.427  mm,	Z =   -242.298  mm,
	W =  90.000 deg,	P =   0.000 deg,	R =   90.000 deg
};
P[2476]{
   GP1:
	UF : 0, UT : 6,		CONFIG : 'N U T, 0, 0, 0',
	X =  273.003  mm,	Y =   -152.224  mm,	Z =   -242.307  mm,
	W =  90.000 deg,	P =   0.000 deg,	R =   90.000 deg
};
P[2477]{
   GP1:
	UF : 0, UT : 6,		CONFIG : 'N U T, 0, 0, 0',
	X =  271.728  mm,	Y =   -152.988  mm,	Z =   -242.376  mm,
	W =  90.000 deg,	P =   0.000 deg,	R =   90.000 deg
};
P[2478]{
   GP1:
	UF : 0, UT : 6,		CONFIG : 'N U T, 0, 0, 0',
	X =  268.396  mm,	Y =   -154.885  mm,	Z =   -242.309  mm,
	W =  90.000 deg,	P =   0.000 deg,	R =   90.000 deg
};
P[2479]{
   GP1:
	UF : 0, UT : 6,		CONFIG : 'N U T, 0, 0, 0',
	X =  266.063  mm,	Y =   -156.152  mm,	Z =   -242.116  mm,
	W =  90.000 deg,	P =   0.000 deg,	R =   90.000 deg
};
P[2480]{
   GP1:
	UF : 0, UT : 6,		CONFIG : 'N U T, 0, 0, 0',
	X =  262.526  mm,	Y =   -158.234  mm,	Z =   -242.212  mm,
	W =  90.000 deg,	P =   0.000 deg,	R =   90.000 deg
};
P[2481]{
   GP1:
	UF : 0, UT : 6,		CONFIG : 'N U T, 0, 0, 0',
	X =  259.199  mm,	Y =   -160.115  mm,	Z =   -242.115  mm,
	W =  90.000 deg,	P =   0.000 deg,	R =   90.000 deg
};
P[2482]{
   GP1:
	UF : 0, UT : 6,		CONFIG : 'N U T, 0, 0, 0',
	X =  257.661  mm,	Y =   -160.916  mm,	Z =   -241.903  mm,
	W =  90.000 deg,	P =   0.000 deg,	R =   90.000 deg
};
P[2483]{
   GP1:
	UF : 0, UT : 6,		CONFIG : 'N U T, 0, 0, 0',
	X =  256.696  mm,	Y =   -161.637  mm,	Z =   -242.301  mm,
	W =  90.000 deg,	P =   0.000 deg,	R =   90.000 deg
};
P[2484]{
   GP1:
	UF : 0, UT : 6,		CONFIG : 'N U T, 0, 0, 0',
	X =  255.495  mm,	Y =   -162.350  mm,	Z =   -242.349  mm,
	W =  90.000 deg,	P =   0.000 deg,	R =   90.000 deg
};
P[2485]{
   GP1:
	UF : 0, UT : 6,		CONFIG : 'N U T, 0, 0, 0',
	X =  254.035  mm,	Y =   -163.105  mm,	Z =   -242.135  mm,
	W =  90.000 deg,	P =   0.000 deg,	R =   90.000 deg
};
P[2486]{
   GP1:
	UF : 0, UT : 6,		CONFIG : 'N U T, 0, 0, 0',
	X =  253.212  mm,	Y =   -163.636  mm,	Z =   -242.272  mm,
	W =  90.000 deg,	P =   0.000 deg,	R =   90.000 deg
};
P[2487]{
   GP1:
	UF : 0, UT : 6,		CONFIG : 'N U T, 0, 0, 0',
	X =  252.586  mm,	Y =   -163.894  mm,	Z =   -242.020  mm,
	W =  90.000 deg,	P =   0.000 deg,	R =   90.000 deg
};
P[2488]{
   GP1:
	UF : 0, UT : 6,		CONFIG : 'N U T, 0, 0, 0',
	X =  248.716  mm,	Y =   -166.167  mm,	Z =   -242.112  mm,
	W =  90.000 deg,	P =   0.000 deg,	R =   90.000 deg
};
P[2489]{
   GP1:
	UF : 0, UT : 6,		CONFIG : 'N U T, 0, 0, 0',
	X =  246.309  mm,	Y =   -167.493  mm,	Z =   -241.960  mm,
	W =  90.000 deg,	P =   0.000 deg,	R =   90.000 deg
};
P[2490]{
   GP1:
	UF : 0, UT : 6,		CONFIG : 'N U T, 0, 0, 0',
	X =  244.175  mm,	Y =   -168.782  mm,	Z =   -242.096  mm,
	W =  90.000 deg,	P =   0.000 deg,	R =   90.000 deg
};
P[2491]{
   GP1:
	UF : 0, UT : 6,		CONFIG : 'N U T, 0, 0, 0',
	X =  243.310  mm,	Y =   -169.340  mm,	Z =   -242.239  mm,
	W =  90.000 deg,	P =   0.000 deg,	R =   90.000 deg
};
P[2492]{
   GP1:
	UF : 0, UT : 6,		CONFIG : 'N U T, 0, 0, 0',
	X =  242.180  mm,	Y =   -169.989  mm,	Z =   -242.229  mm,
	W =  90.000 deg,	P =   0.000 deg,	R =   90.000 deg
};
P[2493]{
   GP1:
	UF : 0, UT : 6,		CONFIG : 'N U T, 0, 0, 0',
	X =  240.811  mm,	Y =   -170.705  mm,	Z =   -242.049  mm,
	W =  90.000 deg,	P =   0.000 deg,	R =   90.000 deg
};
P[2494]{
   GP1:
	UF : 0, UT : 6,		CONFIG : 'N U T, 0, 0, 0',
	X =  239.069  mm,	Y =   -171.729  mm,	Z =   -242.092  mm,
	W =  90.000 deg,	P =   0.000 deg,	R =   90.000 deg
};
P[2495]{
   GP1:
	UF : 0, UT : 6,		CONFIG : 'N U T, 0, 0, 0',
	X =  236.314  mm,	Y =   -173.374  mm,	Z =   -242.224  mm,
	W =  90.000 deg,	P =   0.000 deg,	R =   90.000 deg
};
P[2496]{
   GP1:
	UF : 0, UT : 6,		CONFIG : 'N U T, 0, 0, 0',
	X =  235.429  mm,	Y =   -173.892  mm,	Z =   -242.242  mm,
	W =  90.000 deg,	P =   0.000 deg,	R =   90.000 deg
};
P[2497]{
   GP1:
	UF : 0, UT : 6,		CONFIG : 'N U T, 0, 0, 0',
	X =  234.298  mm,	Y =   -174.531  mm,	Z =   -242.207  mm,
	W =  90.000 deg,	P =   0.000 deg,	R =   90.000 deg
};
P[2498]{
   GP1:
	UF : 0, UT : 6,		CONFIG : 'N U T, 0, 0, 0',
	X =  232.788  mm,	Y =   -175.299  mm,	Z =   -241.956  mm,
	W =  90.000 deg,	P =   0.000 deg,	R =   90.000 deg
};
P[2499]{
   GP1:
	UF : 0, UT : 6,		CONFIG : 'N U T, 0, 0, 0',
	X =  230.718  mm,	Y =   -176.621  mm,	Z =   -242.262  mm,
	W =  90.000 deg,	P =   0.000 deg,	R =   90.000 deg
};
P[2500]{
   GP1:
	UF : 0, UT : 6,		CONFIG : 'N U T, 0, 0, 0',
	X =  226.441  mm,	Y =   -179.088  mm,	Z =   -242.258  mm,
	W =  90.000 deg,	P =   0.000 deg,	R =   90.000 deg
};
P[2501]{
   GP1:
	UF : 0, UT : 6,		CONFIG : 'N U T, 0, 0, 0',
	X =  225.598  mm,	Y =   -179.556  mm,	Z =   -242.211  mm,
	W =  90.000 deg,	P =   0.000 deg,	R =   90.000 deg
};
P[2502]{
   GP1:
	UF : 0, UT : 6,		CONFIG : 'N U T, 0, 0, 0',
	X =  221.306  mm,	Y =   -182.070  mm,	Z =   -242.298  mm,
	W =  90.000 deg,	P =   0.000 deg,	R =   90.000 deg
};
P[2503]{
   GP1:
	UF : 0, UT : 6,		CONFIG : 'N U T, 0, 0, 0',
	X =  215.880  mm,	Y =   -185.159  mm,	Z =   -242.191  mm,
	W =  90.000 deg,	P =   0.000 deg,	R =   90.000 deg
};
P[2504]{
   GP1:
	UF : 0, UT : 6,		CONFIG : 'N U T, 0, 0, 0',
	X =  214.339  mm,	Y =   -186.055  mm,	Z =   -242.208  mm,
	W =  90.000 deg,	P =   0.000 deg,	R =   90.000 deg
};
P[2505]{
   GP1:
	UF : 0, UT : 6,		CONFIG : 'N U T, 0, 0, 0',
	X =  212.715  mm,	Y =   -186.902  mm,	Z =   -241.988  mm,
	W =  90.000 deg,	P =   0.000 deg,	R =   90.000 deg
};
P[2506]{
   GP1:
	UF : 0, UT : 6,		CONFIG : 'N U T, 0, 0, 0',
	X =  211.793  mm,	Y =   -187.554  mm,	Z =   -242.278  mm,
	W =  90.000 deg,	P =   0.000 deg,	R =   90.000 deg
};
P[2507]{
   GP1:
	UF : 0, UT : 6,		CONFIG : 'N U T, 0, 0, 0',
	X =  211.074  mm,	Y =   -187.941  mm,	Z =   -242.208  mm,
	W =  90.000 deg,	P =   0.000 deg,	R =   90.000 deg
};
P[2508]{
   GP1:
	UF : 0, UT : 6,		CONFIG : 'N U T, 0, 0, 0',
	X =  209.020  mm,	Y =   -189.181  mm,	Z =   -242.340  mm,
	W =  90.000 deg,	P =   0.000 deg,	R =   90.000 deg
};
P[2509]{
   GP1:
	UF : 0, UT : 6,		CONFIG : 'N U T, 0, 0, 0',
	X =  208.395  mm,	Y =   -189.539  mm,	Z =   -242.336  mm,
	W =  90.000 deg,	P =   0.000 deg,	R =   90.000 deg
};
P[2510]{
   GP1:
	UF : 0, UT : 6,		CONFIG : 'N U T, 0, 0, 0',
	X =  205.814  mm,	Y =   -190.913  mm,	Z =   -242.051  mm,
	W =  90.000 deg,	P =   0.000 deg,	R =   90.000 deg
};
P[2511]{
   GP1:
	UF : 0, UT : 6,		CONFIG : 'N U T, 0, 0, 0',
	X =  204.653  mm,	Y =   -191.676  mm,	Z =   -242.277  mm,
	W =  90.000 deg,	P =   0.000 deg,	R =   90.000 deg
};
P[2512]{
   GP1:
	UF : 0, UT : 6,		CONFIG : 'N U T, 0, 0, 0',
	X =  199.862  mm,	Y =   -194.416  mm,	Z =   -242.212  mm,
	W =  90.000 deg,	P =   0.000 deg,	R =   90.000 deg
};
P[2513]{
   GP1:
	UF : 0, UT : 6,		CONFIG : 'N U T, 0, 0, 0',
	X =  196.588  mm,	Y =   -196.279  mm,	Z =   -242.146  mm,
	W =  90.000 deg,	P =   0.000 deg,	R =   90.000 deg
};
P[2514]{
   GP1:
	UF : 0, UT : 6,		CONFIG : 'N U T, 0, 0, 0',
	X =  195.853  mm,	Y =   -196.777  mm,	Z =   -242.324  mm,
	W =  90.000 deg,	P =   0.000 deg,	R =   90.000 deg
};
P[2515]{
   GP1:
	UF : 0, UT : 6,		CONFIG : 'N U T, 0, 0, 0',
	X =  194.201  mm,	Y =   -197.646  mm,	Z =   -242.119  mm,
	W =  90.000 deg,	P =   0.000 deg,	R =   90.000 deg
};
P[2516]{
   GP1:
	UF : 0, UT : 6,		CONFIG : 'N U T, 0, 0, 0',
	X =  193.313  mm,	Y =   -198.229  mm,	Z =   -242.288  mm,
	W =  90.000 deg,	P =   0.000 deg,	R =   90.000 deg
};
P[2517]{
   GP1:
	UF : 0, UT : 6,		CONFIG : 'N U T, 0, 0, 0',
	X =  192.070  mm,	Y =   -198.985  mm,	Z =   -242.382  mm,
	W =  90.000 deg,	P =   0.000 deg,	R =   90.000 deg
};
P[2518]{
   GP1:
	UF : 0, UT : 6,		CONFIG : 'N U T, 0, 0, 0',
	X =  189.070  mm,	Y =   -200.530  mm,	Z =   -241.928  mm,
	W =  90.000 deg,	P =   0.000 deg,	R =   90.000 deg
};
P[2519]{
   GP1:
	UF : 0, UT : 6,		CONFIG : 'N U T, 0, 0, 0',
	X =  187.708  mm,	Y =   -201.304  mm,	Z =   -241.897  mm,
	W =  90.000 deg,	P =   0.000 deg,	R =   90.000 deg
};
P[2520]{
   GP1:
	UF : 0, UT : 6,		CONFIG : 'N U T, 0, 0, 0',
	X =  185.710  mm,	Y =   -202.561  mm,	Z =   -242.148  mm,
	W =  90.000 deg,	P =   0.000 deg,	R =   90.000 deg
};
P[2521]{
   GP1:
	UF : 0, UT : 6,		CONFIG : 'N U T, 0, 0, 0',
	X =  184.405  mm,	Y =   -203.208  mm,	Z =   -241.889  mm,
	W =  90.000 deg,	P =   0.000 deg,	R =   90.000 deg
};
P[2522]{
   GP1:
	UF : 0, UT : 6,		CONFIG : 'N U T, 0, 0, 0',
	X =  183.612  mm,	Y =   -203.864  mm,	Z =   -242.370  mm,
	W =  90.000 deg,	P =   0.000 deg,	R =   90.000 deg
};
P[2523]{
   GP1:
	UF : 0, UT : 6,		CONFIG : 'N U T, 0, 0, 0',
	X =  180.171  mm,	Y =   -205.683  mm,	Z =   -241.965  mm,
	W =  90.000 deg,	P =   0.000 deg,	R =   90.000 deg
};
P[2524]{
   GP1:
	UF : 0, UT : 6,		CONFIG : 'N U T, 0, 0, 0',
	X =  179.418  mm,	Y =   -206.181  mm,	Z =   -242.116  mm,
	W =  90.000 deg,	P =   0.000 deg,	R =   90.000 deg
};
P[2525]{
   GP1:
	UF : 0, UT : 6,		CONFIG : 'N U T, 0, 0, 0',
	X =  177.248  mm,	Y =   -207.428  mm,	Z =   -242.105  mm,
	W =  90.000 deg,	P =   0.000 deg,	R =   90.000 deg
};
P[2526]{
   GP1:
	UF : 0, UT : 6,		CONFIG : 'N U T, 0, 0, 0',
	X =  175.442  mm,	Y =   -208.511  mm,	Z =   -242.200  mm,
	W =  90.000 deg,	P =   0.000 deg,	R =   90.000 deg
};
P[2527]{
   GP1:
	UF : 0, UT : 6,		CONFIG : 'N U T, 0, 0, 0',
	X =  174.315  mm,	Y =   -209.097  mm,	Z =   -242.044  mm,
	W =  90.000 deg,	P =   0.000 deg,	R =   90.000 deg
};
P[2528]{
   GP1:
	UF : 0, UT : 6,		CONFIG : 'N U T, 0, 0, 0',
	X =  171.556  mm,	Y =   -210.716  mm,	Z =   -242.109  mm,
	W =  90.000 deg,	P =   0.000 deg,	R =   90.000 deg
};
P[2529]{
   GP1:
	UF : 0, UT : 6,		CONFIG : 'N U T, 0, 0, 0',
	X =  170.928  mm,	Y =   -211.024  mm,	Z =   -241.975  mm,
	W =  90.000 deg,	P =   0.000 deg,	R =   90.000 deg
};
P[2530]{
   GP1:
	UF : 0, UT : 6,		CONFIG : 'N U T, 0, 0, 0',
	X =  168.536  mm,	Y =   -212.407  mm,	Z =   -241.978  mm,
	W =  90.000 deg,	P =   0.000 deg,	R =   90.000 deg
};
P[2531]{
   GP1:
	UF : 0, UT : 6,		CONFIG : 'N U T, 0, 0, 0',
	X =  166.508  mm,	Y =   -213.677  mm,	Z =   -242.218  mm,
	W =  90.000 deg,	P =   0.000 deg,	R =   90.000 deg
};
P[2532]{
   GP1:
	UF : 0, UT : 6,		CONFIG : 'N U T, 0, 0, 0',
	X =  165.157  mm,	Y =   -214.515  mm,	Z =   -242.360  mm,
	W =  90.000 deg,	P =   0.000 deg,	R =   90.000 deg
};
P[2533]{
   GP1:
	UF : 0, UT : 6,		CONFIG : 'N U T, 0, 0, 0',
	X =  163.903  mm,	Y =   -215.053  mm,	Z =   -241.909  mm,
	W =  90.000 deg,	P =   0.000 deg,	R =   90.000 deg
};
P[2534]{
   GP1:
	UF : 0, UT : 6,		CONFIG : 'N U T, 0, 0, 0',
	X =  163.429  mm,	Y =   -215.483  mm,	Z =   -242.290  mm,
	W =  90.000 deg,	P =   0.000 deg,	R =   90.000 deg
};
P[2535]{
   GP1:
	UF : 0, UT : 6,		CONFIG : 'N U T, 0, 0, 0',
	X =  162.666  mm,	Y =   -215.855  mm,	Z =   -242.119  mm,
	W =  90.000 deg,	P =   0.000 deg,	R =   90.000 deg
};
P[2536]{
   GP1:
	UF : 0, UT : 6,		CONFIG : 'N U T, 0, 0, 0',
	X =  161.659  mm,	Y =   -216.494  mm,	Z =   -242.262  mm,
	W =  90.000 deg,	P =   0.000 deg,	R =   90.000 deg
};
P[2537]{
   GP1:
	UF : 0, UT : 6,		CONFIG : 'N U T, 0, 0, 0',
	X =  157.885  mm,	Y =   -218.687  mm,	Z =   -242.294  mm,
	W =  90.000 deg,	P =   0.000 deg,	R =   90.000 deg
};
P[2538]{
   GP1:
	UF : 0, UT : 6,		CONFIG : 'N U T, 0, 0, 0',
	X =  155.695  mm,	Y =   -219.819  mm,	Z =   -241.974  mm,
	W =  90.000 deg,	P =   0.000 deg,	R =   90.000 deg
};
P[2539]{
   GP1:
	UF : 0, UT : 6,		CONFIG : 'N U T, 0, 0, 0',
	X =  153.152  mm,	Y =   -221.375  mm,	Z =   -242.186  mm,
	W =  90.000 deg,	P =   0.000 deg,	R =   90.000 deg
};
P[2540]{
   GP1:
	UF : 0, UT : 6,		CONFIG : 'N U T, 0, 0, 0',
	X =  150.761  mm,	Y =   -222.745  mm,	Z =   -242.160  mm,
	W =  90.000 deg,	P =   0.000 deg,	R =   90.000 deg
};
P[2541]{
   GP1:
	UF : 0, UT : 6,		CONFIG : 'N U T, 0, 0, 0',
	X =  149.162  mm,	Y =   -223.630  mm,	Z =   -242.070  mm,
	W =  90.000 deg,	P =   0.000 deg,	R =   90.000 deg
};
P[2542]{
   GP1:
	UF : 0, UT : 6,		CONFIG : 'N U T, 0, 0, 0',
	X =  147.369  mm,	Y =   -224.720  mm,	Z =   -242.200  mm,
	W =  90.000 deg,	P =   0.000 deg,	R =   90.000 deg
};
P[2543]{
   GP1:
	UF : 0, UT : 6,		CONFIG : 'N U T, 0, 0, 0',
	X =  143.313  mm,	Y =   -227.117  mm,	Z =   -242.334  mm,
	W =  90.000 deg,	P =   0.000 deg,	R =   90.000 deg
};
P[2544]{
   GP1:
	UF : 0, UT : 6,		CONFIG : 'N U T, 0, 0, 0',
	X =  141.553  mm,	Y =   -228.138  mm,	Z =   -242.344  mm,
	W =  90.000 deg,	P =   0.000 deg,	R =   90.000 deg
};
P[2545]{
   GP1:
	UF : 0, UT : 6,		CONFIG : 'N U T, 0, 0, 0',
	X =  139.553  mm,	Y =   -229.211  mm,	Z =   -242.147  mm,
	W =  90.000 deg,	P =   0.000 deg,	R =   90.000 deg
};
P[2546]{
   GP1:
	UF : 0, UT : 6,		CONFIG : 'N U T, 0, 0, 0',
	X =  138.108  mm,	Y =   -230.114  mm,	Z =   -242.313  mm,
	W =  90.000 deg,	P =   0.000 deg,	R =   90.000 deg
};
P[2547]{
   GP1:
	UF : 0, UT : 6,		CONFIG : 'N U T, 0, 0, 0',
	X =  136.694  mm,	Y =   -230.895  mm,	Z =   -242.227  mm,
	W =  90.000 deg,	P =   0.000 deg,	R =   90.000 deg
};
P[2548]{
   GP1:
	UF : 0, UT : 6,		CONFIG : 'N U T, 0, 0, 0',
	X =  134.080  mm,	Y =   -232.376  mm,	Z =   -242.160  mm,
	W =  90.000 deg,	P =   0.000 deg,	R =   90.000 deg
};
P[2549]{
   GP1:
	UF : 0, UT : 6,		CONFIG : 'N U T, 0, 0, 0',
	X =  132.973  mm,	Y =   -233.063  mm,	Z =   -242.277  mm,
	W =  90.000 deg,	P =   0.000 deg,	R =   90.000 deg
};
P[2550]{
   GP1:
	UF : 0, UT : 6,		CONFIG : 'N U T, 0, 0, 0',
	X =  132.033  mm,	Y =   -233.503  mm,	Z =   -242.026  mm,
	W =  90.000 deg,	P =   0.000 deg,	R =   90.000 deg
};
P[2551]{
   GP1:
	UF : 0, UT : 6,		CONFIG : 'N U T, 0, 0, 0',
	X =  128.928  mm,	Y =   -235.377  mm,	Z =   -242.225  mm,
	W =  90.000 deg,	P =   0.000 deg,	R =   90.000 deg
};
P[2552]{
   GP1:
	UF : 0, UT : 6,		CONFIG : 'N U T, 0, 0, 0',
	X =  128.166  mm,	Y =   -235.877  mm,	Z =   -242.371  mm,
	W =  90.000 deg,	P =   0.000 deg,	R =   90.000 deg
};
P[2553]{
   GP1:
	UF : 0, UT : 6,		CONFIG : 'N U T, 0, 0, 0',
	X =  122.744  mm,	Y =   -238.978  mm,	Z =   -242.296  mm,
	W =  90.000 deg,	P =   0.000 deg,	R =   90.000 deg
};
P[2554]{
   GP1:
	UF : 0, UT : 6,		CONFIG : 'N U T, 0, 0, 0',
	X =  121.696  mm,	Y =   -239.550  mm,	Z =   -242.217  mm,
	W =  90.000 deg,	P =   0.000 deg,	R =   90.000 deg
};
P[2555]{
   GP1:
	UF : 0, UT : 6,		CONFIG : 'N U T, 0, 0, 0',
	X =  116.945  mm,	Y =   -242.203  mm,	Z =   -241.997  mm,
	W =  90.000 deg,	P =   0.000 deg,	R =   90.000 deg
};
P[2556]{
   GP1:
	UF : 0, UT : 6,		CONFIG : 'N U T, 0, 0, 0',
	X =  114.524  mm,	Y =   -243.631  mm,	Z =   -242.072  mm,
	W =  90.000 deg,	P =   0.000 deg,	R =   90.000 deg
};
P[2557]{
   GP1:
	UF : 0, UT : 6,		CONFIG : 'N U T, 0, 0, 0',
	X =  112.779  mm,	Y =   -244.624  mm,	Z =   -242.037  mm,
	W =  90.000 deg,	P =   0.000 deg,	R =   90.000 deg
};
P[2558]{
   GP1:
	UF : 0, UT : 6,		CONFIG : 'N U T, 0, 0, 0',
	X =  111.158  mm,	Y =   -245.556  mm,	Z =   -242.026  mm,
	W =  90.000 deg,	P =   0.000 deg,	R =   90.000 deg
};
P[2559]{
   GP1:
	UF : 0, UT : 6,		CONFIG : 'N U T, 0, 0, 0',
	X =  107.642  mm,	Y =   -247.657  mm,	Z =   -242.199  mm,
	W =  90.000 deg,	P =   0.000 deg,	R =   90.000 deg
};
P[2560]{
   GP1:
	UF : 0, UT : 6,		CONFIG : 'N U T, 0, 0, 0',
	X =  106.983  mm,	Y =   -248.080  mm,	Z =   -242.302  mm,
	W =  90.000 deg,	P =   0.000 deg,	R =   90.000 deg
};
P[2561]{
   GP1:
	UF : 0, UT : 6,		CONFIG : 'N U T, 0, 0, 0',
	X =  106.007  mm,	Y =   -248.533  mm,	Z =   -242.033  mm,
	W =  90.000 deg,	P =   0.000 deg,	R =   90.000 deg
};
P[2562]{
   GP1:
	UF : 0, UT : 6,		CONFIG : 'N U T, 0, 0, 0',
	X =  103.998  mm,	Y =   -249.697  mm,	Z =   -242.044  mm,
	W =  90.000 deg,	P =   0.000 deg,	R =   90.000 deg
};
P[2563]{
   GP1:
	UF : 0, UT : 6,		CONFIG : 'N U T, 0, 0, 0',
	X =  101.054  mm,	Y =   -249.009  mm,	Z =   -236.246  mm,
	W =  90.000 deg,	P =   0.000 deg,	R =   90.000 deg
};
P[2564]{
   GP1:
	UF : 0, UT : 6,		CONFIG : 'N U T, 0, 0, 0',
	X =  100.305  mm,	Y =   -249.349  mm,	Z =   -236.023  mm,
	W =  90.000 deg,	P =   0.000 deg,	R =   90.000 deg
};
P[2565]{
   GP1:
	UF : 0, UT : 6,		CONFIG : 'N U T, 0, 0, 0',
	X =  99.750  mm,	Y =   -249.842  mm,	Z =   -236.441  mm,
	W =  90.000 deg,	P =   0.000 deg,	R =   90.000 deg
};
P[2566]{
   GP1:
	UF : 0, UT : 6,		CONFIG : 'N U T, 0, 0, 0',
	X =  97.482  mm,	Y =   -251.000  mm,	Z =   -236.075  mm,
	W =  90.000 deg,	P =   0.000 deg,	R =   90.000 deg
};
P[2567]{
   GP1:
	UF : 0, UT : 6,		CONFIG : 'N U T, 0, 0, 0',
	X =  95.818  mm,	Y =   -252.112  mm,	Z =   -236.441  mm,
	W =  90.000 deg,	P =   0.000 deg,	R =   90.000 deg
};
P[2568]{
   GP1:
	UF : 0, UT : 6,		CONFIG : 'N U T, 0, 0, 0',
	X =  93.986  mm,	Y =   -253.173  mm,	Z =   -236.449  mm,
	W =  90.000 deg,	P =   0.000 deg,	R =   90.000 deg
};
P[2569]{
   GP1:
	UF : 0, UT : 6,		CONFIG : 'N U T, 0, 0, 0',
	X =  91.975  mm,	Y =   -254.287  mm,	Z =   -236.335  mm,
	W =  90.000 deg,	P =   0.000 deg,	R =   90.000 deg
};
P[2570]{
   GP1:
	UF : 0, UT : 6,		CONFIG : 'N U T, 0, 0, 0',
	X =  87.759  mm,	Y =   -256.774  mm,	Z =   -236.464  mm,
	W =  90.000 deg,	P =   0.000 deg,	R =   90.000 deg
};
P[2571]{
   GP1:
	UF : 0, UT : 6,		CONFIG : 'N U T, 0, 0, 0',
	X =  86.224  mm,	Y =   -257.643  mm,	Z =   -236.421  mm,
	W =  90.000 deg,	P =   0.000 deg,	R =   90.000 deg
};
P[2572]{
   GP1:
	UF : 0, UT : 6,		CONFIG : 'N U T, 0, 0, 0',
	X =  84.448  mm,	Y =   -258.549  mm,	Z =   -236.130  mm,
	W =  90.000 deg,	P =   0.000 deg,	R =   90.000 deg
};
P[2573]{
   GP1:
	UF : 0, UT : 6,		CONFIG : 'N U T, 0, 0, 0',
	X =  82.555  mm,	Y =   -259.706  mm,	Z =   -236.287  mm,
	W =  90.000 deg,	P =   0.000 deg,	R =   90.000 deg
};
P[2574]{
   GP1:
	UF : 0, UT : 6,		CONFIG : 'N U T, 0, 0, 0',
	X =  82.015  mm,	Y =   -260.111  mm,	Z =   -236.512  mm,
	W =  90.000 deg,	P =   0.000 deg,	R =   90.000 deg
};
P[2575]{
   GP1:
	UF : 0, UT : 6,		CONFIG : 'N U T, 0, 0, 0',
	X =  78.650  mm,	Y =   -262.025  mm,	Z =   -236.442  mm,
	W =  90.000 deg,	P =   0.000 deg,	R =   90.000 deg
};
P[2576]{
   GP1:
	UF : 0, UT : 6,		CONFIG : 'N U T, 0, 0, 0',
	X =  76.936  mm,	Y =   -263.021  mm,	Z =   -236.457  mm,
	W =  90.000 deg,	P =   0.000 deg,	R =   90.000 deg
};
P[2577]{
   GP1:
	UF : 0, UT : 6,		CONFIG : 'N U T, 0, 0, 0',
	X =  76.024  mm,	Y =   -263.501  mm,	Z =   -236.346  mm,
	W =  90.000 deg,	P =   0.000 deg,	R =   90.000 deg
};
P[2578]{
   GP1:
	UF : 0, UT : 6,		CONFIG : 'N U T, 0, 0, 0',
	X =  74.278  mm,	Y =   -264.472  mm,	Z =   -236.256  mm,
	W =  90.000 deg,	P =   0.000 deg,	R =   90.000 deg
};
P[2579]{
   GP1:
	UF : 0, UT : 6,		CONFIG : 'N U T, 0, 0, 0',
	X =  71.740  mm,	Y =   -265.846  mm,	Z =   -236.034  mm,
	W =  90.000 deg,	P =   0.000 deg,	R =   90.000 deg
};
P[2580]{
   GP1:
	UF : 0, UT : 6,		CONFIG : 'N U T, 0, 0, 0',
	X =  68.701  mm,	Y =   -267.723  mm,	Z =   -236.330  mm,
	W =  90.000 deg,	P =   0.000 deg,	R =   90.000 deg
};
P[2581]{
   GP1:
	UF : 0, UT : 6,		CONFIG : 'N U T, 0, 0, 0',
	X =  66.905  mm,	Y =   -268.763  mm,	Z =   -236.338  mm,
	W =  90.000 deg,	P =   0.000 deg,	R =   90.000 deg
};
P[2582]{
   GP1:
	UF : 0, UT : 6,		CONFIG : 'N U T, 0, 0, 0',
	X =  65.406  mm,	Y =   -269.585  mm,	Z =   -236.228  mm,
	W =  90.000 deg,	P =   0.000 deg,	R =   90.000 deg
};
P[2583]{
   GP1:
	UF : 0, UT : 6,		CONFIG : 'N U T, 0, 0, 0',
	X =  64.799  mm,	Y =   -269.985  mm,	Z =   -236.351  mm,
	W =  90.000 deg,	P =   0.000 deg,	R =   90.000 deg
};
P[2584]{
   GP1:
	UF : 0, UT : 6,		CONFIG : 'N U T, 0, 0, 0',
	X =  64.236  mm,	Y =   -270.338  mm,	Z =   -236.419  mm,
	W =  90.000 deg,	P =   0.000 deg,	R =   90.000 deg
};
P[2585]{
   GP1:
	UF : 0, UT : 6,		CONFIG : 'N U T, 0, 0, 0',
	X =  59.732  mm,	Y =   -272.968  mm,	Z =   -236.489  mm,
	W =  90.000 deg,	P =   0.000 deg,	R =   90.000 deg
};
P[2586]{
   GP1:
	UF : 0, UT : 6,		CONFIG : 'N U T, 0, 0, 0',
	X =  57.064  mm,	Y =   -274.480  mm,	Z =   -236.422  mm,
	W =  90.000 deg,	P =   0.000 deg,	R =   90.000 deg
};
P[2587]{
   GP1:
	UF : 0, UT : 6,		CONFIG : 'N U T, 0, 0, 0',
	X =  56.290  mm,	Y =   -274.858  mm,	Z =   -236.254  mm,
	W =  90.000 deg,	P =   0.000 deg,	R =   90.000 deg
};
P[2588]{
   GP1:
	UF : 0, UT : 6,		CONFIG : 'N U T, 0, 0, 0',
	X =  55.531  mm,	Y =   -275.355  mm,	Z =   -236.397  mm,
	W =  90.000 deg,	P =   0.000 deg,	R =   90.000 deg
};
P[2589]{
   GP1:
	UF : 0, UT : 6,		CONFIG : 'N U T, 0, 0, 0',
	X =  54.219  mm,	Y =   -276.070  mm,	Z =   -236.292  mm,
	W =  90.000 deg,	P =   0.000 deg,	R =   90.000 deg
};
P[2590]{
   GP1:
	UF : 0, UT : 6,		CONFIG : 'N U T, 0, 0, 0',
	X =  51.598  mm,	Y =   -277.625  mm,	Z =   -236.393  mm,
	W =  90.000 deg,	P =   0.000 deg,	R =   90.000 deg
};
P[2591]{
   GP1:
	UF : 0, UT : 6,		CONFIG : 'N U T, 0, 0, 0',
	X =  46.580  mm,	Y =   -280.540  mm,	Z =   -236.438  mm,
	W =  90.000 deg,	P =   0.000 deg,	R =   90.000 deg
};
P[2592]{
   GP1:
	UF : 0, UT : 6,		CONFIG : 'N U T, 0, 0, 0',
	X =  41.948  mm,	Y =   -283.218  mm,	Z =   -236.444  mm,
	W =  90.000 deg,	P =   0.000 deg,	R =   90.000 deg
};
P[2593]{
   GP1:
	UF : 0, UT : 6,		CONFIG : 'N U T, 0, 0, 0',
	X =  40.361  mm,	Y =   -284.103  mm,	Z =   -236.370  mm,
	W =  90.000 deg,	P =   0.000 deg,	R =   90.000 deg
};
P[2594]{
   GP1:
	UF : 0, UT : 6,		CONFIG : 'N U T, 0, 0, 0',
	X =  34.449  mm,	Y =   -287.432  mm,	Z =   -236.164  mm,
	W =  90.000 deg,	P =   0.000 deg,	R =   90.000 deg
};
P[2595]{
   GP1:
	UF : 0, UT : 6,		CONFIG : 'N U T, 0, 0, 0',
	X =  33.557  mm,	Y =   -288.008  mm,	Z =   -236.314  mm,
	W =  90.000 deg,	P =   0.000 deg,	R =   90.000 deg
};
P[2596]{
   GP1:
	UF : 0, UT : 6,		CONFIG : 'N U T, 0, 0, 0',
	X =  30.342  mm,	Y =   -289.837  mm,	Z =   -236.246  mm,
	W =  90.000 deg,	P =   0.000 deg,	R =   90.000 deg
};
P[2597]{
   GP1:
	UF : 0, UT : 6,		CONFIG : 'N U T, 0, 0, 0',
	X =  26.417  mm,	Y =   -292.192  mm,	Z =   -236.460  mm,
	W =  90.000 deg,	P =   0.000 deg,	R =   90.000 deg
};
P[2598]{
   GP1:
	UF : 0, UT : 6,		CONFIG : 'N U T, 0, 0, 0',
	X =  24.281  mm,	Y =   -293.352  mm,	Z =   -236.284  mm,
	W =  90.000 deg,	P =   0.000 deg,	R =   90.000 deg
};
P[2599]{
   GP1:
	UF : 0, UT : 6,		CONFIG : 'N U T, 0, 0, 0',
	X =  21.351  mm,	Y =   -294.936  mm,	Z =   -236.022  mm,
	W =  90.000 deg,	P =   0.000 deg,	R =   90.000 deg
};
P[2600]{
   GP1:
	UF : 0, UT : 6,		CONFIG : 'N U T, 0, 0, 0',
	X =  20.617  mm,	Y =   -295.537  mm,	Z =   -236.451  mm,
	W =  90.000 deg,	P =   0.000 deg,	R =   90.000 deg
};
P[2601]{
   GP1:
	UF : 0, UT : 6,		CONFIG : 'N U T, 0, 0, 0',
	X =  19.883  mm,	Y =   -295.943  mm,	Z =   -236.408  mm,
	W =  90.000 deg,	P =   0.000 deg,	R =   90.000 deg
};
P[2602]{
   GP1:
	UF : 0, UT : 6,		CONFIG : 'N U T, 0, 0, 0',
	X =  18.349  mm,	Y =   -296.738  mm,	Z =   -236.190  mm,
	W =  90.000 deg,	P =   0.000 deg,	R =   90.000 deg
};
P[2603]{
   GP1:
	UF : 0, UT : 6,		CONFIG : 'N U T, 0, 0, 0',
	X =  15.827  mm,	Y =   -298.247  mm,	Z =   -236.317  mm,
	W =  90.000 deg,	P =   0.000 deg,	R =   90.000 deg
};
P[2604]{
   GP1:
	UF : 0, UT : 6,		CONFIG : 'N U T, 0, 0, 0',
	X =  14.944  mm,	Y =   -298.698  mm,	Z =   -236.175  mm,
	W =  90.000 deg,	P =   0.000 deg,	R =   90.000 deg
};
P[2605]{
   GP1:
	UF : 0, UT : 6,		CONFIG : 'N U T, 0, 0, 0',
	X =  14.314  mm,	Y =   -299.095  mm,	Z =   -236.256  mm,
	W =  90.000 deg,	P =   0.000 deg,	R =   90.000 deg
};
P[2606]{
   GP1:
	UF : 0, UT : 6,		CONFIG : 'N U T, 0, 0, 0',
	X =  11.620  mm,	Y =   -300.687  mm,	Z =   -236.343  mm,
	W =  90.000 deg,	P =   0.000 deg,	R =   90.000 deg
};
P[2607]{
   GP1:
	UF : 0, UT : 6,		CONFIG : 'N U T, 0, 0, 0',
	X =  10.820  mm,	Y =   -301.096  mm,	Z =   -236.217  mm,
	W =  90.000 deg,	P =   0.000 deg,	R =   90.000 deg
};
P[2608]{
   GP1:
	UF : 0, UT : 6,		CONFIG : 'N U T, 0, 0, 0',
	X =  10.222  mm,	Y =   -301.527  mm,	Z =   -236.421  mm,
	W =  90.000 deg,	P =   0.000 deg,	R =   90.000 deg
};
P[2609]{
   GP1:
	UF : 0, UT : 6,		CONFIG : 'N U T, 0, 0, 0',
	X =  6.283  mm,	Y =   -303.638  mm,	Z =   -236.026  mm,
	W =  90.000 deg,	P =   0.000 deg,	R =   90.000 deg
};
P[2610]{
   GP1:
	UF : 0, UT : 6,		CONFIG : 'N U T, 0, 0, 0',
	X =  2.862  mm,	Y =   -305.738  mm,	Z =   -236.328  mm,
	W =  90.000 deg,	P =   0.000 deg,	R =   90.000 deg
};
P[2611]{
   GP1:
	UF : 0, UT : 6,		CONFIG : 'N U T, 0, 0, 0',
	X =  2.242  mm,	Y =   -305.987  mm,	Z =   -236.065  mm,
	W =  90.000 deg,	P =   0.000 deg,	R =   90.000 deg
};
P[2612]{
   GP1:
	UF : 0, UT : 6,		CONFIG : 'N U T, 0, 0, 0',
	X =  1.617  mm,	Y =   -306.468  mm,	Z =   -236.357  mm,
	W =  90.000 deg,	P =   0.000 deg,	R =   90.000 deg
};
P[2613]{
   GP1:
	UF : 0, UT : 6,		CONFIG : 'N U T, 0, 0, 0',
	X =  0.599  mm,	Y =   -306.997  mm,	Z =   -236.212  mm,
	W =  90.000 deg,	P =   0.000 deg,	R =   90.000 deg
};
P[2614]{
   GP1:
	UF : 0, UT : 6,		CONFIG : 'N U T, 0, 0, 0',
	X =  -0.848  mm,	Y =   -307.893  mm,	Z =   -236.362  mm,
	W =  90.000 deg,	P =   0.000 deg,	R =   90.000 deg
};
P[2615]{
   GP1:
	UF : 0, UT : 6,		CONFIG : 'N U T, 0, 0, 0',
	X =  -2.228  mm,	Y =   -308.693  mm,	Z =   -236.369  mm,
	W =  90.000 deg,	P =   0.000 deg,	R =   90.000 deg
};
P[2616]{
   GP1:
	UF : 0, UT : 6,		CONFIG : 'N U T, 0, 0, 0',
	X =  -6.487  mm,	Y =   -311.151  mm,	Z =   -236.368  mm,
	W =  90.000 deg,	P =   0.000 deg,	R =   90.000 deg
};
P[2617]{
   GP1:
	UF : 0, UT : 6,		CONFIG : 'N U T, 0, 0, 0',
	X =  -8.889  mm,	Y =   -312.485  mm,	Z =   -236.236  mm,
	W =  90.000 deg,	P =   0.000 deg,	R =   90.000 deg
};
P[2618]{
   GP1:
	UF : 0, UT : 6,		CONFIG : 'N U T, 0, 0, 0',
	X =  -10.443  mm,	Y =   -313.430  mm,	Z =   -236.353  mm,
	W =  90.000 deg,	P =   0.000 deg,	R =   90.000 deg
};
P[2619]{
   GP1:
	UF : 0, UT : 6,		CONFIG : 'N U T, 0, 0, 0',
	X =  -12.580  mm,	Y =   -314.679  mm,	Z =   -236.389  mm,
	W =  90.000 deg,	P =   0.000 deg,	R =   90.000 deg
};
P[2620]{
   GP1:
	UF : 0, UT : 6,		CONFIG : 'N U T, 0, 0, 0',
	X =  -15.569  mm,	Y =   -316.268  mm,	Z =   -236.058  mm,
	W =  90.000 deg,	P =   0.000 deg,	R =   90.000 deg
};
P[2621]{
   GP1:
	UF : 0, UT : 6,		CONFIG : 'N U T, 0, 0, 0',
	X =  -16.720  mm,	Y =   -317.009  mm,	Z =   -236.243  mm,
	W =  90.000 deg,	P =   0.000 deg,	R =   90.000 deg
};
P[2622]{
   GP1:
	UF : 0, UT : 6,		CONFIG : 'N U T, 0, 0, 0',
	X =  -20.066  mm,	Y =   -319.045  mm,	Z =   -236.496  mm,
	W =  90.000 deg,	P =   0.000 deg,	R =   90.000 deg
};
P[2623]{
   GP1:
	UF : 0, UT : 6,		CONFIG : 'N U T, 0, 0, 0',
	X =  -23.934  mm,	Y =   -321.209  mm,	Z =   -236.328  mm,
	W =  90.000 deg,	P =   0.000 deg,	R =   90.000 deg
};
P[2624]{
   GP1:
	UF : 0, UT : 6,		CONFIG : 'N U T, 0, 0, 0',
	X =  -24.772  mm,	Y =   -321.686  mm,	Z =   -236.314  mm,
	W =  90.000 deg,	P =   0.000 deg,	R =   90.000 deg
};
P[2625]{
   GP1:
	UF : 0, UT : 6,		CONFIG : 'N U T, 0, 0, 0',
	X =  -26.637  mm,	Y =   -322.720  mm,	Z =   -236.209  mm,
	W =  90.000 deg,	P =   0.000 deg,	R =   90.000 deg
};
P[2626]{
   GP1:
	UF : 0, UT : 6,		CONFIG : 'N U T, 0, 0, 0',
	X =  -27.239  mm,	Y =   -322.989  mm,	Z =   -236.017  mm,
	W =  90.000 deg,	P =   0.000 deg,	R =   90.000 deg
};
P[2627]{
   GP1:
	UF : 0, UT : 6,		CONFIG : 'N U T, 0, 0, 0',
	X =  -28.240  mm,	Y =   -323.748  mm,	Z =   -236.453  mm,
	W =  90.000 deg,	P =   0.000 deg,	R =   90.000 deg
};
P[2628]{
   GP1:
	UF : 0, UT : 6,		CONFIG : 'N U T, 0, 0, 0',
	X =  -29.593  mm,	Y =   -324.477  mm,	Z =   -236.329  mm,
	W =  90.000 deg,	P =   0.000 deg,	R =   90.000 deg
};
P[2629]{
   GP1:
	UF : 0, UT : 6,		CONFIG : 'N U T, 0, 0, 0',
	X =  -33.470  mm,	Y =   -326.678  mm,	Z =   -236.237  mm,
	W =  90.000 deg,	P =   0.000 deg,	R =   90.000 deg
};
P[2630]{
   GP1:
	UF : 0, UT : 6,		CONFIG : 'N U T, 0, 0, 0',
	X =  -34.590  mm,	Y =   -327.298  mm,	Z =   -236.173  mm,
	W =  90.000 deg,	P =   0.000 deg,	R =   90.000 deg
};
P[2631]{
   GP1:
	UF : 0, UT : 6,		CONFIG : 'N U T, 0, 0, 0',
	X =  -36.641  mm,	Y =   -328.543  mm,	Z =   -236.320  mm,
	W =  90.000 deg,	P =   0.000 deg,	R =   90.000 deg
};
P[2632]{
   GP1:
	UF : 0, UT : 6,		CONFIG : 'N U T, 0, 0, 0',
	X =  -37.449  mm,	Y =   -328.970  mm,	Z =   -236.223  mm,
	W =  90.000 deg,	P =   0.000 deg,	R =   90.000 deg
};
P[2633]{
   GP1:
	UF : 0, UT : 6,		CONFIG : 'N U T, 0, 0, 0',
	X =  -39.294  mm,	Y =   -330.043  mm,	Z =   -236.244  mm,
	W =  90.000 deg,	P =   0.000 deg,	R =   90.000 deg
};
P[2634]{
   GP1:
	UF : 0, UT : 6,		CONFIG : 'N U T, 0, 0, 0',
	X =  -44.305  mm,	Y =   -332.952  mm,	Z =   -236.281  mm,
	W =  90.000 deg,	P =   0.000 deg,	R =   90.000 deg
};
P[2635]{
   GP1:
	UF : 0, UT : 6,		CONFIG : 'N U T, 0, 0, 0',
	X =  -45.830  mm,	Y =   -333.905  mm,	Z =   -236.457  mm,
	W =  90.000 deg,	P =   0.000 deg,	R =   90.000 deg
};
P[2636]{
   GP1:
	UF : 0, UT : 6,		CONFIG : 'N U T, 0, 0, 0',
	X =  -46.945  mm,	Y =   -334.523  mm,	Z =   -236.395  mm,
	W =  90.000 deg,	P =   0.000 deg,	R =   90.000 deg
};
P[2637]{
   GP1:
	UF : 0, UT : 6,		CONFIG : 'N U T, 0, 0, 0',
	X =  -48.377  mm,	Y =   -335.352  mm,	Z =   -236.401  mm,
	W =  90.000 deg,	P =   0.000 deg,	R =   90.000 deg
};
P[2638]{
   GP1:
	UF : 0, UT : 6,		CONFIG : 'N U T, 0, 0, 0',
	X =  -50.442  mm,	Y =   -336.530  mm,	Z =   -236.365  mm,
	W =  90.000 deg,	P =   0.000 deg,	R =   90.000 deg
};
P[2639]{
   GP1:
	UF : 0, UT : 6,		CONFIG : 'N U T, 0, 0, 0',
	X =  -51.250  mm,	Y =   -336.892  mm,	Z =   -236.112  mm,
	W =  90.000 deg,	P =   0.000 deg,	R =   90.000 deg
};
P[2640]{
   GP1:
	UF : 0, UT : 6,		CONFIG : 'N U T, 0, 0, 0',
	X =  -51.989  mm,	Y =   -337.342  mm,	Z =   -236.166  mm,
	W =  90.000 deg,	P =   0.000 deg,	R =   90.000 deg
};
P[2641]{
   GP1:
	UF : 0, UT : 6,		CONFIG : 'N U T, 0, 0, 0',
	X =  -53.238  mm,	Y =   -338.009  mm,	Z =   -236.039  mm,
	W =  90.000 deg,	P =   0.000 deg,	R =   90.000 deg
};
P[2642]{
   GP1:
	UF : 0, UT : 6,		CONFIG : 'N U T, 0, 0, 0',
	X =  -54.472  mm,	Y =   -338.837  mm,	Z =   -236.317  mm,
	W =  90.000 deg,	P =   0.000 deg,	R =   90.000 deg
};
P[2643]{
   GP1:
	UF : 0, UT : 6,		CONFIG : 'N U T, 0, 0, 0',
	X =  -58.736  mm,	Y =   -341.357  mm,	Z =   -236.458  mm,
	W =  90.000 deg,	P =   0.000 deg,	R =   90.000 deg
};
P[2644]{
   GP1:
	UF : 0, UT : 6,		CONFIG : 'N U T, 0, 0, 0',
	X =  -59.598  mm,	Y =   -341.811  mm,	Z =   -236.353  mm,
	W =  90.000 deg,	P =   0.000 deg,	R =   90.000 deg
};
P[2645]{
   GP1:
	UF : 0, UT : 6,		CONFIG : 'N U T, 0, 0, 0',
	X =  -60.460  mm,	Y =   -342.251  mm,	Z =   -236.213  mm,
	W =  90.000 deg,	P =   0.000 deg,	R =   90.000 deg
};
P[2646]{
   GP1:
	UF : 0, UT : 6,		CONFIG : 'N U T, 0, 0, 0',
	X =  -61.368  mm,	Y =   -342.742  mm,	Z =   -236.131  mm,
	W =  90.000 deg,	P =   0.000 deg,	R =   90.000 deg
};
P[2647]{
   GP1:
	UF : 0, UT : 6,		CONFIG : 'N U T, 0, 0, 0',
	X =  -62.190  mm,	Y =   -343.373  mm,	Z =   -236.511  mm,
	W =  90.000 deg,	P =   0.000 deg,	R =   90.000 deg
};
P[2648]{
   GP1:
	UF : 0, UT : 6,		CONFIG : 'N U T, 0, 0, 0',
	X =  -62.954  mm,	Y =   -343.781  mm,	Z =   -236.429  mm,
	W =  90.000 deg,	P =   0.000 deg,	R =   90.000 deg
};
P[2649]{
   GP1:
	UF : 0, UT : 6,		CONFIG : 'N U T, 0, 0, 0',
	X =  -63.975  mm,	Y =   -344.322  mm,	Z =   -236.314  mm,
	W =  90.000 deg,	P =   0.000 deg,	R =   90.000 deg
};
P[2650]{
   GP1:
	UF : 0, UT : 6,		CONFIG : 'N U T, 0, 0, 0',
	X =  -67.883  mm,	Y =   -346.524  mm,	Z =   -236.180  mm,
	W =  90.000 deg,	P =   0.000 deg,	R =   90.000 deg
};
P[2651]{
   GP1:
	UF : 0, UT : 6,		CONFIG : 'N U T, 0, 0, 0',
	X =  -69.913  mm,	Y =   -347.783  mm,	Z =   -236.392  mm,
	W =  90.000 deg,	P =   0.000 deg,	R =   90.000 deg
};
P[2652]{
   GP1:
	UF : 0, UT : 6,		CONFIG : 'N U T, 0, 0, 0',
	X =  -74.258  mm,	Y =   -350.340  mm,	Z =   -236.507  mm,
	W =  90.000 deg,	P =   0.000 deg,	R =   90.000 deg
};
P[2653]{
   GP1:
	UF : 0, UT : 6,		CONFIG : 'N U T, 0, 0, 0',
	X =  -79.226  mm,	Y =   -353.100  mm,	Z =   -236.245  mm,
	W =  90.000 deg,	P =   0.000 deg,	R =   90.000 deg
};
P[2654]{
   GP1:
	UF : 0, UT : 6,		CONFIG : 'N U T, 0, 0, 0',
	X =  -80.377  mm,	Y =   -353.836  mm,	Z =   -236.420  mm,
	W =  90.000 deg,	P =   0.000 deg,	R =   90.000 deg
};
P[2655]{
   GP1:
	UF : 0, UT : 6,		CONFIG : 'N U T, 0, 0, 0',
	X =  -81.318  mm,	Y =   -354.335  mm,	Z =   -236.309  mm,
	W =  90.000 deg,	P =   0.000 deg,	R =   90.000 deg
};
P[2656]{
   GP1:
	UF : 0, UT : 6,		CONFIG : 'N U T, 0, 0, 0',
	X =  -83.403  mm,	Y =   -355.602  mm,	Z =   -236.463  mm,
	W =  90.000 deg,	P =   0.000 deg,	R =   90.000 deg
};
P[2657]{
   GP1:
	UF : 0, UT : 6,		CONFIG : 'N U T, 0, 0, 0',
	X =  -85.633  mm,	Y =   -356.902  mm,	Z =   -236.494  mm,
	W =  90.000 deg,	P =   0.000 deg,	R =   90.000 deg
};
P[2658]{
   GP1:
	UF : 0, UT : 6,		CONFIG : 'N U T, 0, 0, 0',
	X =  -88.090  mm,	Y =   -358.282  mm,	Z =   -236.400  mm,
	W =  90.000 deg,	P =   0.000 deg,	R =   90.000 deg
};
P[2659]{
   GP1:
	UF : 0, UT : 6,		CONFIG : 'N U T, 0, 0, 0',
	X =  -90.366  mm,	Y =   -359.482  mm,	Z =   -236.122  mm,
	W =  90.000 deg,	P =   0.000 deg,	R =   90.000 deg
};
P[2660]{
   GP1:
	UF : 0, UT : 6,		CONFIG : 'N U T, 0, 0, 0',
	X =  -92.217  mm,	Y =   -360.538  mm,	Z =   -236.093  mm,
	W =  90.000 deg,	P =   0.000 deg,	R =   90.000 deg
};
P[2661]{
   GP1:
	UF : 0, UT : 6,		CONFIG : 'N U T, 0, 0, 0',
	X =  -92.878  mm,	Y =   -361.030  mm,	Z =   -236.359  mm,
	W =  90.000 deg,	P =   0.000 deg,	R =   90.000 deg
};
P[2662]{
   GP1:
	UF : 0, UT : 6,		CONFIG : 'N U T, 0, 0, 0',
	X =  -96.229  mm,	Y =   -362.912  mm,	Z =   -236.231  mm,
	W =  90.000 deg,	P =   0.000 deg,	R =   90.000 deg
};
P[2663]{
   GP1:
	UF : 0, UT : 6,		CONFIG : 'N U T, 0, 0, 0',
	X =  -98.967  mm,	Y =   -364.568  mm,	Z =   -236.413  mm,
	W =  90.000 deg,	P =   0.000 deg,	R =   90.000 deg
};
P[2664]{
   GP1:
	UF : 0, UT : 6,		CONFIG : 'N U T, 0, 0, 0',
	X =  -101.936  mm,	Y =   -366.264  mm,	Z =   -236.371  mm,
	W =  90.000 deg,	P =   0.000 deg,	R =   90.000 deg
};
P[2665]{
   GP1:
